(* CODESYS project SeltZVU3.project

Project tree, tasks and I/O mapping:
  Device : Owen SPK1xx, Owen, order no. 023, version 3.5.4.20
    application Application
      libraries: Standard, * (System); CmpSysExec, 1.0.0.2 (Owen); SysTime, * (System); VisuDialogs, * (System); Util, * (System); CAA File, * (CAA Technical Workgroup)
      task MainTask (cyclic, interval t#10ms, priority 1) calls PLC_PRG
      task VISU_TASK (cyclic, interval t#100ms, priority 31) calls VisuElems.Visu_Prg
      task Task_ZAKALKA (cyclic, interval t#10ms, priority 1) calls ZAKALKA
      task READ_WRITE_ZAKALKA_PROG (cyclic, interval t#10ms, priority 1) calls WRITE_PROGRAM_FILE_ON_SD, READ_PROGRAM_FROM_FILE
      task Archivating (cyclic, interval t#10ms, priority 1) calls Archive
      task Task_TransmitingFiles (cyclic, interval t#10ms, priority 1) calls READ_FILE_ON_SD, WRITE_FILE_ON_SD
      task ConnectWithComputer (cyclic, interval t#10ms, priority 1) calls MB_PC
      program PLC_PRG [ST]
      program ClearBuf [ST]
      program DataPrepare [ST]
      program RD_param [ST]
      program READ_PROGRAM_FROM_FILE [ST]: Analyz_str, Find_Symbol
      global variables GVL
      program ZAKALKA [ST]
      program SearchFile [ST]
      text list Modbus_Error_list
      text list Status_v_Rabote
      text list Warning_Text_list
      visualisation Archive_manager
      visualisation Center_indukt
      visualisation KeypadNumpad
      visualisation Modbus_param
      visualisation Regim_choice
      visualisation Zakalka_program
      visualisation Zakalka_work
      program WRITE_PROGRAM_FILE_ON_SD [ST]
      program Archive [ST]: Archivation, make_log_collection, Work_with_Flash
      program WRITE_FILE_ON_SD [ST]
      program READ_FILE_ON_SD [ST]
    SLAVE_COM : Modbus COM, 3S - Smart Software Solutions GmbH, version 3.4.0.0
        settings: DataBits = 8; StopBits = 1; ComPort = 3
      MB_PC : Modbus Serial Device, 3S - Smart Software Solutions GmbH, version 3.5.5.0
          input  Application.buffer_name_file[0] : WORD  // Inputs.Inputs
          input  Application.buffer_name_file[1] : WORD  // Inputs.Inputs
          input  Application.buffer_name_file[2] : WORD  // Inputs.Inputs
          input  Application.buffer_name_file[3] : WORD  // Inputs.Inputs
          input  Application.buffer_name_file[4] : WORD  // Inputs.Inputs
          input  Application.buffer_name_file[5] : WORD  // Inputs.Inputs
          input  Application.buffer_name_file[6] : WORD  // Inputs.Inputs
          input  Application.buffer_name_file[7] : WORD  // Inputs.Inputs
          input  Application.buffer_name_file[8] : WORD  // Inputs.Inputs
          input  Application.buffer_name_file[9] : WORD  // Inputs.Inputs
          input  Application.buffer_name_file[10] : WORD  // Inputs.Inputs
          input  Application.buffer_name_file[11] : WORD  // Inputs.Inputs
          input  Application.buffer_name_file[12] : WORD  // Inputs.Inputs
          input  Application.buffer_name_file[13] : WORD  // Inputs.Inputs
          input  Application.buffer_name_file[14] : WORD  // Inputs.Inputs
          input  Application.buffer_name_file[15] : WORD  // Inputs.Inputs
          input  Application.buffer_name_file[16] : WORD  // Inputs.Inputs
          input  Application.buffer_name_file[17] : WORD  // Inputs.Inputs
          input  Application.buffer_name_file[18] : WORD  // Inputs.Inputs
          input  Application.buffer_name_file[19] : WORD  // Inputs.Inputs
          input  Application.buffer_name_file[20] : WORD  // Inputs.Inputs
          input  Application.buffer_name_file[21] : WORD  // Inputs.Inputs
          input  Application.buffer_name_file[22] : WORD  // Inputs.Inputs
          input  Application.buffer_name_file[23] : WORD  // Inputs.Inputs
          input  Application.buffer_name_file[24] : WORD  // Inputs.Inputs
          input  Application.buffer_wr[0] : WORD  // Inputs.Inputs
          input  Application.buffer_wr[1] : WORD  // Inputs.Inputs
          input  Application.buffer_wr[2] : WORD  // Inputs.Inputs
          input  Application.buffer_wr[3] : WORD  // Inputs.Inputs
          input  Application.buffer_wr[4] : WORD  // Inputs.Inputs
          input  Application.buffer_wr[5] : WORD  // Inputs.Inputs
          input  Application.buffer_wr[6] : WORD  // Inputs.Inputs
          input  Application.buffer_wr[7] : WORD  // Inputs.Inputs
          input  Application.buffer_wr[8] : WORD  // Inputs.Inputs
          input  Application.buffer_wr[9] : WORD  // Inputs.Inputs
          input  Application.buffer_wr[10] : WORD  // Inputs.Inputs
          input  Application.buffer_wr[11] : WORD  // Inputs.Inputs
          input  Application.buffer_wr[12] : WORD  // Inputs.Inputs
          input  Application.buffer_wr[13] : WORD  // Inputs.Inputs
          input  Application.buffer_wr[14] : WORD  // Inputs.Inputs
          input  Application.buffer_wr[15] : WORD  // Inputs.Inputs
          input  Application.buffer_wr[16] : WORD  // Inputs.Inputs
          input  Application.buffer_wr[17] : WORD  // Inputs.Inputs
          input  Application.buffer_wr[18] : WORD  // Inputs.Inputs
          input  Application.buffer_wr[19] : WORD  // Inputs.Inputs
          input  Application.buffer_wr[20] : WORD  // Inputs.Inputs
          input  Application.buffer_wr[21] : WORD  // Inputs.Inputs
          input  Application.buffer_wr[22] : WORD  // Inputs.Inputs
          input  Application.buffer_wr[23] : WORD  // Inputs.Inputs
          input  Application.buffer_wr[24] : WORD  // Inputs.Inputs
          input  Application.buffer_wr[25] : WORD  // Inputs.Inputs
          input  Application.buffer_wr[26] : WORD  // Inputs.Inputs
          input  Application.buffer_wr[27] : WORD  // Inputs.Inputs
          input  Application.buffer_wr[28] : WORD  // Inputs.Inputs
          input  Application.buffer_wr[29] : WORD  // Inputs.Inputs
          input  Application.buffer_wr[30] : WORD  // Inputs.Inputs
          input  Application.buffer_wr[31] : WORD  // Inputs.Inputs
          input  Application.buffer_wr[32] : WORD  // Inputs.Inputs
          input  Application.buffer_wr[33] : WORD  // Inputs.Inputs
          input  Application.buffer_wr[34] : WORD  // Inputs.Inputs
          input  Application.buffer_wr[35] : WORD  // Inputs.Inputs
          input  Application.buffer_wr[36] : WORD  // Inputs.Inputs
          input  Application.buffer_wr[37] : WORD  // Inputs.Inputs
          input  Application.buffer_wr[38] : WORD  // Inputs.Inputs
          input  Application.buffer_wr[39] : WORD  // Inputs.Inputs
          input  Application.buffer_wr[40] : WORD  // Inputs.Inputs
          input  Application.buffer_wr[41] : WORD  // Inputs.Inputs
          input  Application.buffer_wr[42] : WORD  // Inputs.Inputs
          input  Application.buffer_wr[43] : WORD  // Inputs.Inputs
          input  Application.buffer_wr[44] : WORD  // Inputs.Inputs
          input  Application.buffer_wr[45] : WORD  // Inputs.Inputs
          input  Application.buffer_wr[46] : WORD  // Inputs.Inputs
          input  Application.buffer_wr[47] : WORD  // Inputs.Inputs
          input  Application.buffer_wr[48] : WORD  // Inputs.Inputs
          input  Application.buffer_wr[49] : WORD  // Inputs.Inputs
          input  Application.buffer_wr[50] : WORD  // Inputs.Inputs
          input  Application.buffer_wr[51] : WORD  // Inputs.Inputs
          input  Application.buffer_wr[52] : WORD  // Inputs.Inputs
          input  Application.buffer_wr[53] : WORD  // Inputs.Inputs
          input  Application.buffer_wr[54] : WORD  // Inputs.Inputs
          input  Application.buffer_wr[55] : WORD  // Inputs.Inputs
          input  Application.buffer_wr[56] : WORD  // Inputs.Inputs
          input  Application.buffer_wr[57] : WORD  // Inputs.Inputs
          input  Application.buffer_wr[58] : WORD  // Inputs.Inputs
          input  Application.buffer_wr[59] : WORD  // Inputs.Inputs
          input  Application.buffer_wr[60] : WORD  // Inputs.Inputs
          input  Application.buffer_wr[61] : WORD  // Inputs.Inputs
          input  Application.buffer_wr[62] : WORD  // Inputs.Inputs
          input  Application.buffer_wr[63] : WORD  // Inputs.Inputs
          input  Application.buffer_wr[64] : WORD  // Inputs.Inputs
          input  Application.buffer_wr[65] : WORD  // Inputs.Inputs
          input  Application.buffer_wr[66] : WORD  // Inputs.Inputs
          input  Application.buffer_wr[67] : WORD  // Inputs.Inputs
          input  Application.buffer_wr[68] : WORD  // Inputs.Inputs
          input  Application.buffer_wr[69] : WORD  // Inputs.Inputs
          input  Application.buffer_wr[70] : WORD  // Inputs.Inputs
          input  Application.buffer_wr[71] : WORD  // Inputs.Inputs
          input  Application.buffer_wr[72] : WORD  // Inputs.Inputs
          input  Application.buffer_wr[73] : WORD  // Inputs.Inputs
          input  Application.buffer_wr[74] : WORD  // Inputs.Inputs
          input  Application.buffer_wr[75] : WORD  // Inputs.Inputs
          input  Application.buffer_wr[76] : WORD  // Inputs.Inputs
          input  Application.buffer_wr[77] : WORD  // Inputs.Inputs
          input  Application.buffer_wr[78] : WORD  // Inputs.Inputs
          input  Application.buffer_wr[79] : WORD  // Inputs.Inputs
          input  Application.buffer_wr[80] : WORD  // Inputs.Inputs
          input  Application.buffer_wr[81] : WORD  // Inputs.Inputs
          input  Application.buffer_wr[82] : WORD  // Inputs.Inputs
          input  Application.buffer_wr[83] : WORD  // Inputs.Inputs
          input  Application.buffer_wr[84] : WORD  // Inputs.Inputs
          input  Application.buffer_wr[85] : WORD  // Inputs.Inputs
          input  Application.buffer_wr[86] : WORD  // Inputs.Inputs
          input  Application.buffer_wr[87] : WORD  // Inputs.Inputs
          input  Application.buffer_wr[88] : WORD  // Inputs.Inputs
          input  Application.buffer_wr[89] : WORD  // Inputs.Inputs
          input  Application.buffer_wr[90] : WORD  // Inputs.Inputs
          input  Application.buffer_wr[91] : WORD  // Inputs.Inputs
          input  Application.buffer_wr[92] : WORD  // Inputs.Inputs
          input  Application.buffer_wr[93] : WORD  // Inputs.Inputs
          input  Application.buffer_wr[94] : WORD  // Inputs.Inputs
          input  Application.buffer_wr[95] : WORD  // Inputs.Inputs
          input  Application.buffer_wr[96] : WORD  // Inputs.Inputs
          input  Application.buffer_wr[97] : WORD  // Inputs.Inputs
          input  Application.buffer_wr[98] : WORD  // Inputs.Inputs
          input  Application.buffer_wr[99] : WORD  // Inputs.Inputs
          input  Application.buffer_wr[100] : WORD  // Inputs.Inputs
          input  Application.buffer_wr[101] : WORD  // Inputs.Inputs
          input  Application.buffer_wr[102] : WORD  // Inputs.Inputs
          input  Application.buffer_wr[103] : WORD  // Inputs.Inputs
          input  Application.buffer_wr[104] : WORD  // Inputs.Inputs
          input  Application.buffer_wr[105] : WORD  // Inputs.Inputs
          input  Application.buffer_wr[106] : WORD  // Inputs.Inputs
          input  Application.buffer_wr[107] : WORD  // Inputs.Inputs
          input  Application.buffer_wr[108] : WORD  // Inputs.Inputs
          input  Application.buffer_wr[109] : WORD  // Inputs.Inputs
          input  Application.buffer_wr[110] : WORD  // Inputs.Inputs
          input  Application.buffer_wr[111] : WORD  // Inputs.Inputs
          input  Application.buffer_wr[112] : WORD  // Inputs.Inputs
          input  Application.buffer_wr[113] : WORD  // Inputs.Inputs
          input  Application.buffer_wr[114] : WORD  // Inputs.Inputs
          input  Application.buffer_wr[115] : WORD  // Inputs.Inputs
          input  Application.buffer_wr[116] : WORD  // Inputs.Inputs
          input  Application.buffer_wr[117] : WORD  // Inputs.Inputs
          input  Application.buffer_wr[118] : WORD  // Inputs.Inputs
          input  Application.buffer_wr[119] : WORD  // Inputs.Inputs
          input  Application.buffer_wr[120] : WORD  // Inputs.Inputs
          input  Application.WRITE_FILE_ON_SD.size_block : WORD  // Inputs.Inputs
          input  Application.WRITE_FILE_ON_SD.START_STOP_WRITE : WORD  // Inputs.Inputs
          input  Application.READ_FILE_ON_SD.START_STOP_READ : WORD  // Inputs.Inputs
          input  Application.PLC_PRG.SCAN_SD_START_STOP : WORD  // Inputs.Inputs
          input  Application.READ_FILE_ON_SD.RESET_FUNC : WORD  // Inputs.Inputs
          output Application.READ_FILE_ON_SD.SIZE_LR : WORD  // Outputs.Outputs
          output Application.READ_FILE_ON_SD.SIZE_HR : WORD  // Outputs.Outputs
          output Application.buffer[0] : WORD  // Outputs.Outputs
          output Application.buffer[1] : WORD  // Outputs.Outputs
          output Application.buffer[2] : WORD  // Outputs.Outputs
          output Application.buffer[3] : WORD  // Outputs.Outputs
          output Application.buffer[4] : WORD  // Outputs.Outputs
          output Application.buffer[5] : WORD  // Outputs.Outputs
          output Application.buffer[6] : WORD  // Outputs.Outputs
          output Application.buffer[7] : WORD  // Outputs.Outputs
          output Application.buffer[8] : WORD  // Outputs.Outputs
          output Application.buffer[9] : WORD  // Outputs.Outputs
          output Application.buffer[10] : WORD  // Outputs.Outputs
          output Application.buffer[11] : WORD  // Outputs.Outputs
          output Application.buffer[12] : WORD  // Outputs.Outputs
          output Application.buffer[13] : WORD  // Outputs.Outputs
          output Application.buffer[14] : WORD  // Outputs.Outputs
          output Application.buffer[15] : WORD  // Outputs.Outputs
          output Application.buffer[16] : WORD  // Outputs.Outputs
          output Application.buffer[17] : WORD  // Outputs.Outputs
          output Application.buffer[18] : WORD  // Outputs.Outputs
          output Application.buffer[19] : WORD  // Outputs.Outputs
          output Application.buffer[20] : WORD  // Outputs.Outputs
          output Application.buffer[21] : WORD  // Outputs.Outputs
          output Application.buffer[22] : WORD  // Outputs.Outputs
          output Application.buffer[23] : WORD  // Outputs.Outputs
          output Application.buffer[24] : WORD  // Outputs.Outputs
          output Application.buffer[25] : WORD  // Outputs.Outputs
          output Application.buffer[26] : WORD  // Outputs.Outputs
          output Application.buffer[27] : WORD  // Outputs.Outputs
          output Application.buffer[28] : WORD  // Outputs.Outputs
          output Application.buffer[29] : WORD  // Outputs.Outputs
          output Application.buffer[30] : WORD  // Outputs.Outputs
          output Application.buffer[31] : WORD  // Outputs.Outputs
          output Application.buffer[32] : WORD  // Outputs.Outputs
          output Application.buffer[33] : WORD  // Outputs.Outputs
          output Application.buffer[34] : WORD  // Outputs.Outputs
          output Application.buffer[35] : WORD  // Outputs.Outputs
          output Application.buffer[36] : WORD  // Outputs.Outputs
          output Application.buffer[37] : WORD  // Outputs.Outputs
          output Application.buffer[38] : WORD  // Outputs.Outputs
          output Application.buffer[39] : WORD  // Outputs.Outputs
          output Application.buffer[40] : WORD  // Outputs.Outputs
          output Application.buffer[41] : WORD  // Outputs.Outputs
          output Application.buffer[42] : WORD  // Outputs.Outputs
          output Application.buffer[43] : WORD  // Outputs.Outputs
          output Application.buffer[44] : WORD  // Outputs.Outputs
          output Application.buffer[45] : WORD  // Outputs.Outputs
          output Application.buffer[46] : WORD  // Outputs.Outputs
          output Application.buffer[47] : WORD  // Outputs.Outputs
          output Application.buffer[48] : WORD  // Outputs.Outputs
          output Application.buffer[49] : WORD  // Outputs.Outputs
          output Application.buffer[50] : WORD  // Outputs.Outputs
          output Application.buffer[51] : WORD  // Outputs.Outputs
          output Application.buffer[52] : WORD  // Outputs.Outputs
          output Application.buffer[53] : WORD  // Outputs.Outputs
          output Application.buffer[54] : WORD  // Outputs.Outputs
          output Application.buffer[55] : WORD  // Outputs.Outputs
          output Application.buffer[56] : WORD  // Outputs.Outputs
          output Application.buffer[57] : WORD  // Outputs.Outputs
          output Application.buffer[58] : WORD  // Outputs.Outputs
          output Application.buffer[59] : WORD  // Outputs.Outputs
          output Application.buffer[60] : WORD  // Outputs.Outputs
          output Application.buffer[61] : WORD  // Outputs.Outputs
          output Application.buffer[62] : WORD  // Outputs.Outputs
          output Application.buffer[63] : WORD  // Outputs.Outputs
          output Application.buffer[64] : WORD  // Outputs.Outputs
          output Application.buffer[65] : WORD  // Outputs.Outputs
          output Application.buffer[66] : WORD  // Outputs.Outputs
          output Application.buffer[67] : WORD  // Outputs.Outputs
          output Application.buffer[68] : WORD  // Outputs.Outputs
          output Application.buffer[69] : WORD  // Outputs.Outputs
          output Application.buffer[70] : WORD  // Outputs.Outputs
          output Application.buffer[71] : WORD  // Outputs.Outputs
          output Application.buffer[72] : WORD  // Outputs.Outputs
          output Application.buffer[73] : WORD  // Outputs.Outputs
          output Application.buffer[74] : WORD  // Outputs.Outputs
          output Application.buffer[75] : WORD  // Outputs.Outputs
          output Application.buffer[76] : WORD  // Outputs.Outputs
          output Application.buffer[77] : WORD  // Outputs.Outputs
          output Application.buffer[78] : WORD  // Outputs.Outputs
          output Application.buffer[79] : WORD  // Outputs.Outputs
          output Application.buffer[80] : WORD  // Outputs.Outputs
          output Application.buffer[81] : WORD  // Outputs.Outputs
          output Application.buffer[82] : WORD  // Outputs.Outputs
          output Application.buffer[83] : WORD  // Outputs.Outputs
          output Application.buffer[84] : WORD  // Outputs.Outputs
          output Application.buffer[85] : WORD  // Outputs.Outputs
          output Application.buffer[86] : WORD  // Outputs.Outputs
          output Application.buffer[87] : WORD  // Outputs.Outputs
          output Application.buffer[88] : WORD  // Outputs.Outputs
          output Application.buffer[89] : WORD  // Outputs.Outputs
          output Application.buffer[90] : WORD  // Outputs.Outputs
          output Application.buffer[91] : WORD  // Outputs.Outputs
          output Application.buffer[92] : WORD  // Outputs.Outputs
          output Application.buffer[93] : WORD  // Outputs.Outputs
          output Application.buffer[94] : WORD  // Outputs.Outputs
          output Application.buffer[95] : WORD  // Outputs.Outputs
          output Application.buffer[96] : WORD  // Outputs.Outputs
          output Application.buffer[97] : WORD  // Outputs.Outputs
          output Application.buffer[98] : WORD  // Outputs.Outputs
          output Application.buffer[99] : WORD  // Outputs.Outputs
          output Application.buffer[100] : WORD  // Outputs.Outputs
          output Application.buffer[101] : WORD  // Outputs.Outputs
          output Application.buffer[102] : WORD  // Outputs.Outputs
          output Application.buffer[103] : WORD  // Outputs.Outputs
          output Application.buffer[104] : WORD  // Outputs.Outputs
          output Application.buffer[105] : WORD  // Outputs.Outputs
          output Application.buffer[106] : WORD  // Outputs.Outputs
          output Application.buffer[107] : WORD  // Outputs.Outputs
          output Application.buffer[108] : WORD  // Outputs.Outputs
          output Application.buffer[109] : WORD  // Outputs.Outputs
          output Application.buffer[110] : WORD  // Outputs.Outputs
          output Application.buffer[111] : WORD  // Outputs.Outputs
          output Application.buffer[112] : WORD  // Outputs.Outputs
          output Application.buffer[113] : WORD  // Outputs.Outputs
          output Application.buffer[114] : WORD  // Outputs.Outputs
          output Application.buffer[115] : WORD  // Outputs.Outputs
          output Application.buffer[116] : WORD  // Outputs.Outputs
          output Application.buffer[117] : WORD  // Outputs.Outputs
          output Application.buffer[118] : WORD  // Outputs.Outputs
          output Application.buffer[119] : WORD  // Outputs.Outputs
          output Application.buffer[120] : WORD  // Outputs.Outputs
          output Application.buffer[121] : WORD  // Outputs.Outputs
          output Application.buffer[122] : WORD  // Outputs.Outputs
          output Application.buffer[123] : WORD  // Outputs.Outputs
          output Application.buffer[124] : WORD  // Outputs.Outputs
          output Application.WRITE_FILE_ON_SD.CycleWriteDone : WORD  // Outputs.Outputs
          output Application.FileError : WORD  // Outputs.Outputs
          output Application.READ_FILE_ON_SD.RESET_SUC : BOOL  // Outputs.Outputs.Bit0
          output Application.READ_FILE_ON_SD.cnt_cycle : WORD  // Outputs.Outputs
          unmapped channels: Inputs, Outputs
    Modbus_COM : Modbus COM, 3S - Smart Software Solutions GmbH, version 3.4.0.0
        settings: DataBits = 8; StopBits = 1; ComPort = 2
      Modbus_Master_COM_Port : Modbus Master, COM Port, 3S - Smart Software Solutions GmbH, version 3.5.5.0
          settings: Transmission = 'RTU'; ResponseTimeout = 500; TimeBetweenFrames = 50; Auto-restart communication = TRUE
        Modbus_Slave_Atxmega128 : Modbus Slave, COM Port, 3S - Smart Software Solutions GmbH, version 3.5.4.0
            settings: SlaveAddress = 9; ResponseTimeout = 500; UseExtendedFunctionCodes = TRUE; Channel7.Function Code = 3; Channel7.Read Offset = 16#0000; Channel7.Read Length = 51; Channel7.Write Offset = 0; Channel7.Write Length = 0; Channel7.Cycle Time = 500; To_Atxmega_KN_NACHALO.Function Code = 16; To_Atxmega_KN_NACHALO.Read Offset = 0; To_Atxmega_KN_NACHALO.Read Length = 0; To_Atxmega_KN_NACHALO.Write Offset = 16#0032; To_Atxmega_KN_NACHALO.Write Length = 1; To_Atxmega_KN_NACHALO.Cycle Time = 500; Channel 2.Function Code = 4; Channel 2.Read Offset = 16#0000; Channel 2.Read Length = 23; Channel 2.Write Offset = 0; Channel 2.Write Length = 0; Channel 2.Cycle Time = 500; Channel 3.Function Code = 16; Channel 3.Read Offset = 0; Channel 3.Read Length = 0; Channel 3.Write Offset = 16#0001; Channel 3.Write Length = 12; Channel 3.Cycle Time = 100; Channel 6.Function Code = 6; Channel 6.Read Offset = 0; Channel 6.Read Length = 0; Channel 6.Write Offset = 16#0000; Channel 6.Write Length = 1; Channel 6.Cycle Time = 100; Channel 5.Function Code = 16; Channel 5.Read Offset = 0; Channel 5.Read Length = 0; Channel 5.Write Offset = 16#0033; Channel 5.Write Length = 123; Channel 5.Cycle Time = 100
            input  Application.PLC_PRG.DY_start : WORD  // Channel7.Channel7
            input  Application.ZAKALKA.opros_DY_kn_nachalo : BOOL  // Channel7.Channel7.Bit0
            output Application.PLC_PRG.DY_kn_nachalo : BOOL  // To_Atxmega_KN_NACHALO.To_Atxmega_KN_NACHALO.Bit0
            input  Application.PLC_PRG.PORTKH : WORD  // Channel 2.Channel 2
            input  Application.PLC_PRG.PORTCF : WORD  // Channel 2.Channel 2
            input  Application.PLC_PRG.WarningText_mod : WORD  // Channel 2.Channel 2
            input  Application.t_prog_LCD : WORD  // Channel 2.Channel 2
            input  Application.W_schet_vat : WORD  // Channel 2.Channel 2
            input  Application.zona : WORD  // Channel 2.Channel 2
            input  Application.P_ind : WORD  // Channel 2.Channel 2
            input  Application.T_rad_max : WORD  // Channel 2.Channel 2
            input  Application.zona_reg : WORD  // Channel 2.Channel 2
            input  Application.n_nagrev : WORD  // Channel 2.Channel 2
            input  Application.i_t_regim : WORD  // Channel 2.Channel 2
            input  Application.Frec_LCD_point : WORD  // Channel 2.Channel 2
            input  Application.U_pit_max : WORD  // Channel 2.Channel 2
            input  Application.tekyheePosition_lcd : WORD  // Channel 2.Channel 2
            input  Application.I_lcd : WORD  // Channel 2.Channel 2
            input  Application.zadachaPosition_lcd : WORD  // Channel 2.Channel 2
            output Application.PLC_PRG.UP_DOWN : WORD  // Channel 3.Channel 3
            output Application.DistRegim : WORD  // Channel 3.Channel 3
            output Application.PLC_PRG.MB_4_20_kanal_1 : WORD  // Channel 3.Channel 3
            output Application.PLC_PRG.MB_4_20_kanal_2 : WORD  // Channel 3.Channel 3
            output Application.ZAKALKA.zakalka_nachalo : WORD  // Channel 3.Channel 3
            output Application.ZAKALKA.rotation_on : BOOL  // Channel 3.Channel 3.Bit0
            output Application.ZAKALKA.spreer_prednagrev : BOOL  // Channel 3.Channel 3.Bit0
            output Application.ZAKALKA.diagnostik : BOOL  // Channel 3.Channel 3.Bit0
            output Application.ZAKALKA.OTPUSK : BOOL  // Channel 3.Channel 3.Bit0
            output Application.L_peremesh_ohl : WORD  // Channel 3.Channel 3
            output Application.PLC_PRG.b_req_start_stop : BIT  // Channel 6
            output Application.PLC_PRG.CMD_start : ARRAY[0..0] OF WORD  // Channel 6
            output Application.PLC_PRG.Req_WR_Params : BIT  // Channel 5
            output Application.PLC_PRG.Buffer : ARRAY[0..122] OF WORD  // Channel 5
            unmapped channels: Channel7, To_Atxmega_KN_NACHALO, Channel 2, Channel 3
        Modbus_Slave_MY110 : Modbus Slave, COM Port, 3S - Smart Software Solutions GmbH, version 3.5.4.0
            settings: SlaveAddress = 16; ResponseTimeout = 500; UseExtendedFunctionCodes = TRUE; Channel 0.Function Code = 15; Channel 0.Read Offset = 0; Channel 0.Read Length = 0; Channel 0.Write Offset = 16#0000; Channel 0.Write Length = 8; Channel 0.Cycle Time = 250
            output Application.PLC_PRG.ZAGIM_UP : BOOL  // Channel 0.Channel 0.Bit0
            output Application.PLC_PRG.ZAGIM_DOWN : BOOL  // Channel 0.Channel 0.Bit1
            output Application.PLC_PRG.CENTER_DOWN : BOOL  // Channel 0.Channel 0.Bit2
            output Application.PLC_PRG.CENTER_UP : BOOL  // Channel 0.Channel 0.Bit3
            output Application.PLC_PRG.DET_CIRCLE_ON : BOOL  // Channel 0.Channel 0.Bit4
            output Application.PLC_PRG.SPREER_ON : BOOL  // Channel 0.Channel 0.Bit5
            output Application.PLC_PRG.CENTER_LEFT : BOOL  // Channel 0.Channel 0.Bit6
            output Application.PLC_PRG.CENTER_RIGHT : BOOL  // Channel 0.Channel 0.Bit7
            unmapped channels: Channel 0
  text list GlobalTextList
  text list NachaloVerhNiz
*)

// Device/Application/GVL
VAR_GLOBAL
	ProgramFiles:STRING(255):='/mnt/ufs/media/mmcblk0p1/ProgramFiles/';
	ArchiveFiles:STRING(255):='/mnt/ufs/media/mmcblk0p1/Archive/';		
	nomer_zoni: ARRAY [1..20] OF INT;
	zona_rabochaya: USINT := 1;	
	
	(*Датчики*)
	PORTK: BYTE;
	PORTH: BYTE;
	PORTC: BYTE;
	PORTF: BYTE;
	
	WarningText: WORD := 1;
	t_prog_LCD: WORD;
	W_schet_vat: WORD;
	zona : WORD;
	P_ind: WORD;
	T_rad_max: WORD;
	zona_reg: WORD;
	n_nagrev: WORD;
	R_ind_lcd: WORD; 
	i_t_regim: WORD := 3;
	DistRegim: WORD;
	DY_gotovn : BOOL;
	Frec_LCD: WORD;
	U_pit_max: WORD;
	U_pit_min: WORD;
 	tekyheePosition_lcd: WORD;
	Frec_LCD_point:WORD;
	h_faza:WORD;
	I_lcd:WORD;
	zadachaPosition_lcd: WORD;
	
	rotation_on: BOOL; 
	
	buffer: ARRAY[0..125] OF WORD;
	buffer_name_file: ARRAY [0..24] OF WORD;
	buffer_wr: ARRAY[0..120] OF WORD;
	
	FileError: INT;//Ошибка при записи файла по модбасу
	ExError	: BOOL;
	StrError : STRING(255);
	READING: BOOL;
	WRITING: BOOL;
	RESET_ERROR:BOOL;
	
(*	OTPUSK_P_nachaln_nagrev: ARRAY [1..10] OF INT;
	OTPUSK_t_nachaln_nagrev: ARRAY [1..10] OF INT;
	OTPUSK_P_nagrev: ARRAY [1..10] OF INT;
	OTPUSK_V_peremeshenia: ARRAY [1..10] OF BYTE;
	OTPUSK_t_freeze: ARRAY [1..10] OF INT;*)
	
END_VAR

VAR_GLOBAL PERSISTENT RETAIN
	chislo_zon: WORD := 1;
//	Nachalo: INT;//Зачем убрал из параметров для хранения в ПЗУ ?	
	P_nachaln_nagrev: ARRAY [1..20] OF INT;//Мощность на преднагрев
	t_nachaln_nagrev: ARRAY [1..20] OF INT;//Время а преднагрев
	P_nagrev: ARRAY [1..20] OF INT;//Мощность в движени
	L_peremeshenia: ARRAY [1..20] OF INT;//Длиназоны
	V_peremeshenia: ARRAY [1..20] OF INT;//Сорость пермщеия
	t_freeze: ARRAY [1..20] OF INT;//Вемя охлаждения
	L_to_next_zone: ARRAY [1..20] OF INT;//Растояние до слдующейзоны
	L_peremesh_ohl: WORD;
END_VAR

// Device/Application/PLC_PRG
PROGRAM PLC_PRG

VAR_INPUT
	ReqStart : BOOL := FALSE; //Запрос на старт при нажатие кнопок старт = 1 после отправки запроса = 0
	Req_WR_Params : BOOL := FALSE; //запрос на передачу параметров в МК
	Req_OverWriting_param : BOOL := FALSE;
	DY_start: WORD;//отображает состояние кнопок старт/стоп и состояние МК
	CMD_start: WORD;//1-Старт 0-Стоп
	Req_START_STOP: BOOL;//Запрос на передачу команды старт/стоп
	DY_kn_nachalo: BOOL := FALSE; //кнопка начало 0-неактивна 1-актив
END_VAR

VAR
	Timer_Req_WR_params:TON;
	Timer_Inc_Speed:TON;
	TMR_START:TON;
	b_req_start_stop:BOOL;//Тригер для передачи команды старт стоп
	MB_4_20_kanal_2 : INT:=7000;//Скорость вращения нижнего центра
	MB_4_20_kanal_1 : INT:=7000;//Скорость перемещения индуктора/детали	
	
	PORTKH: WORD;
	PORTCF: WORD;
	ReqStop : BOOL := FALSE; //Запрос на стоп при нажатие кнопок стоп = 1 после отправки запроса = 0
	
	UP_DOWN : WORD := 0; // верх вниз 0-стоп 1-в верх 2-в низ
	
 
	START: BOOL := FALSE; //старт установки
	STOP: BOOL := TRUE; //стоп установки
	
	CENTER_UP: BOOL;
	CENTER_DOWN: BOOL;
	CENTER_LEFT: BOOL;
	CENTER_RIGHT: BOOL;
	ZAGIM_UP: BOOL;
	ZAGIM_DOWN: BOOL;
	DET_CIRCLE_ON: BOOL;	//вкл вращение
	DET_CIRCLE_SPIN: BOOL; //вкл регулирование скорости
	DET_CIRCLE_SPEED: WORD; //скорость вращения детали
	SPREER_ON: BOOL;
	
	Buffer : ARRAY[0..122] OF WORD;
	cmpl: BOOL;
	err: INT;
	TimeOut : TIME:=T#300MS;
	DataSize : WORD;
	Connect : BOOL :=FALSE;
	master : BYTE := 3;
	CNT_REG : BYTE;
	
	(*Входные параметры*)
	in1: BOOL;
	in2: BOOL; 
	in3: BOOL;//Датчик низа
	in4: BOOL;
	in5: BOOL;
	in6: BOOL;//Датчик верха
	in7: BOOL;
	in8: BOOL;
	in9: BOOL;
	in10: BOOL;//Кнопка начало
	in11: BOOL;
	
	TEMP  : WORD;  
	(*конец входные параметры*)
	
	Button: WORD;
	ButAddr: WORD;
	
	WarningText_mod: WORD;
	Butt_UP: BOOL;
	Butt_DOWN: BOOL;
	
	//Время
	result_time: UDINT;
	time_dword: DWORD;
	time_of_st: DATE_AND_TIME;
	
	Symbols: ARRAY[0..4] OF BYTE;
	stroka:STRING;
	p_str:POINTER TO BYTE;
	i:BYTE;
	
	(*Работа с файловой системой*)
	SCAN_SD_START_STOP:WORD;
	ErrorModbus_Atxmega: IoDrvModbus.MB_ErrorCodes;
	ErrorModbus_MY110: INT;
END_VAR

PORTK := WORD_TO_BYTE(SHR(PORTKH,8));
PORTH := WORD_TO_BYTE(PORTKH);
PORTC := WORD_TO_BYTE(SHR(PORTCF,8));
PORTF := WORD_TO_BYTE(PORTCF);
in1 := NOT(GVL.PORTK.4);
in2 := GVL.PORTK.5;
in3 := GVL.PORTK.6;
in4 := GVL.PORTK.7;
in5 := GVL.PORTH.3;
in6 := GVL.PORTH.2;
in7 := GVL.PORTC.2;
in8 := GVL.PORTC.3;
in9 := GVL.PORTC.4;
in10:= GVL.PORTC.5;
in11:= GVL.PORTF.6;

IF CMD_start=DY_start=1 THEN
	Req_START_STOP:=FALSE;
END_IF

TMR_START(IN:=Req_START_STOP,PT:=T#50MS);
IF TMR_START.Q THEN
	TMR_START(IN:=FALSE);
	b_req_start_stop:=NOT(b_req_start_stop);
END_IF

Timer_Req_WR_params(IN:=DY_kn_nachalo OR Req_OverWriting_param, PT:=T#200MS , Q=> , ET=> );
IF Timer_Req_WR_params.Q THEN //(DY_kn_nachalo OR Req_OverWriting_param) AND (cnt_timer>30)THEN
	DataPrepare(chislo_zon:=GVL.chislo_zon,P_nachaln_nagrev:=GVL.P_nachaln_nagrev,t_nachaln_nagrev:=GVL.t_nachaln_nagrev,P_nagrev:=GVL.P_nagrev,V_peremeshenia:=GVL.V_peremeshenia,L_peremeshenia:=GVL.L_peremeshenia,L_to_next_zone:=GVL.L_to_next_zone,t_freeze:=GVL.t_freeze, Buffer=>Buffer);
	Timer_Req_WR_params(IN:=FALSE);
//	DY_kn_nachalo:=FALSE;
	Req_OverWriting_param:=FALSE;
	Req_WR_Params:=TRUE;
END_IF

Timer_Inc_Speed(IN:=((UP_DOWN=2) OR (UP_DOWN=1)), PT:=T#100MS , Q=> , ET=> );
IF Timer_Inc_Speed.Q THEN //(DY_kn_nachalo OR Req_OverWriting_param) AND (cnt_timer>30)THEN
	Timer_Inc_Speed(IN:=FALSE);
	IF MB_4_20_kanal_1  + 100 >= 20000 THEN
		MB_4_20_kanal_1:=20000;	
	ELSE
		MB_4_20_kanal_1:=MB_4_20_kanal_1+100;	
	END_IF
END_IF

IF UP_DOWN=0 THEN
	MB_4_20_kanal_1:=7000;
END_IF

IF dy_start = 1 THEN
	VisuElems.CurrentVisu:='Zakalka_work';
END_IF

IF (dy_start = 0) AND (VisuElems.CurrentVisu = 'Zakalka_work') THEN
	VisuElems.CurrentVisu := 'Zakalka_program';
END_IF

time_dword:=SysTimeRtcGet(pResult:=result_time );
time_of_st:=DWORD_TO_DT(time_dword);

ErrorModbus_Atxmega := Modbus_Slave_Atxmega128.byModbusError;
ErrorModbus_MY110 := Modbus_Slave_MY110.byModbusError;

END_PROGRAM

// Device/Application/DataPrepare
PROGRAM DataPrepare
VAR_INPUT
	chislo_zon: WORD;
	P_nachaln_nagrev: ARRAY [1..20] OF INT;
	t_nachaln_nagrev: ARRAY [1..20] OF INT;
	P_nagrev: ARRAY [1..20] OF INT;
	V_peremeshenia: ARRAY [1..20] OF INT;
	L_peremeshenia: ARRAY [1..20] OF INT;
	L_to_next_zone: ARRAY [1..20] OF INT;
	t_freeze: ARRAY [1..20] OF INT;
END_VAR

VAR_OUTPUT
	Buffer: ARRAY[0..122] OF WORD;
END_VAR

VAR
	TEMP: INT;
	Counter: INT;
	index: INT;
	knopka_nachalo: BYTE :=1;
END_VAR

index:=0;
Buffer[index]:= chislo_zon;
index:=index+1;
	
FOR Counter:=(1+ZAKALKA.shift_otpusk) TO (chislo_zon+ZAKALKA.shift_otpusk) BY 1 DO
	Buffer[index]:= t_nachaln_nagrev[Counter];
	index:=index+1;
	
	Buffer[index]:= p_nachaln_nagrev[Counter];
	index:=index+1;
	
	Buffer[index]:= V_peremeshenia[Counter];
	index:=index+1;
	

	Buffer[index]:= L_peremeshenia[Counter-ZAKALKA.shift_otpusk];
	index:=index+1;


	Buffer[index]:= P_nagrev[Counter];
	index:=index+1;
	
	
	Buffer[index]:= t_freeze[Counter];
	index:=index+1;
	
	Buffer[index]:= L_to_next_zone[Counter-ZAKALKA.shift_otpusk];
	index:=index+1;
END_FOR

END_PROGRAM

// Device/Application/ZAKALKA
PROGRAM ZAKALKA
VAR
Zakalochniy_cikl: INT;
stage: INT := 1;	
AutoCicleFinish:WORD;

Zakalka_otpusk_active: BOOL := TRUE; //выбран ярлык редактирования отпуска
L_between_stels: BOOL := TRUE;
i_zona: USINT := 1; //заполнитель кнопки зона
OTPUSK: BOOL;//Запуск отпуска


shift_otpusk: INT;
Zakalka_last_zona: BOOL;
color_indukt: DWORD;

pressed_find_prog:BOOL;//true когда нажата кнопка найти программу
pressed_create_new_prog:BOOL;
enter_value:BOOL;//true - при закрытии клавы по кнопке OK
SearchThroughArray: STRING;//Имя файла для поиска существующей программы закалки
new_prog: STRING;//Имя файла для новой программы 
result_prog: ARRAY [1..10] OF STRING(255);//Результаты поиска
	i_result_prog: INT :=1;//Активный размер масива result_prog
enter_prog: INT:=1;//Индекс выбранной программы в массиве result_prog
buf_enter_prog : INT:=1;//Предыдущее значение enter_prog
test_ok: BOOL :=FALSE;
	opros_DY_kn_nachalo: BOOL;
update_drop_list:BOOL;
	buf_size_list:INT;//предыдущая длина списка найденных файлов
END_VAR

VAR_INPUT
	Otpusk_on: BOOL;//отпуск включен
	Zakalka_on: BOOL:=TRUE;
 	spreer_prednagrev: BOOL;
	diagnostik: BOOL:=TRUE;
	rotation_on: BOOL:=TRUE; 
	
	zakalka_nachalo: INT;
END_VAR
VAR_OUTPUT

END_VAR

IF PLC_PRG.DY_start=1 THEN
	Archive.arch_en:=TRUE;
ELSE	
	Archive.arch_en:=FALSE;
END_IF

IF (PLC_PRG.DY_kn_nachalo) AND (opros_DY_kn_nachalo = TRUE) THEN
	PLC_PRG.DY_kn_nachalo := FALSE;
END_IF

IF (Otpusk_on <> TRUE) THEN
	Zakalka_otpusk_active := TRUE;
ELSE
	IF (ZAKALKA.Zakalka_on <> TRUE) THEN
	Zakalka_otpusk_active := FALSE;
	END_IF
END_IF

IF (zona_rabochaya = chislo_zon) THEN
	Zakalka_last_zona := TRUE;
ELSE
	Zakalka_last_zona := FALSE;
END_IF


IF PLC_PRG.DY_start = 0  AND ((ZAKALKA.stage <> 3 AND ZAKALKA.stage <> 2) OR (PLC_PRG.WarningText_mod = 53)) THEN
	ZAKALKA.stage := 0;
	
	IF (ZAKALKA.Zakalka_on) AND (ZAKALKA.Otpusk_on = FALSE) THEN //цикл закалка без отпуска
		ZAKALKA.Zakalochniy_cikl := 1;
		shift_otpusk := 0;
		OTPUSK := FALSE;
	END_IF
	
	IF (ZAKALKA.Zakalka_on = FALSE) AND (ZAKALKA.Otpusk_on) THEN //цикл отпуск без закалки
		ZAKALKA.Zakalochniy_cikl := 2;
		shift_otpusk := 10;
		OTPUSK := TRUE;
	END_IF
	
	IF (ZAKALKA.Zakalka_on) AND (ZAKALKA.Otpusk_on) THEN		//цикл закалка с отпуском
		ZAKALKA.Zakalochniy_cikl := 3;
		shift_otpusk := 0;
		OTPUSK := FALSE;
	END_IF
		PLC_PRG.Req_WR_Params := FALSE;
		PLC_PRG.Req_OverWriting_param := TRUE;
END_IF

IF PLC_PRG.DY_start = 1  AND ZAKALKA.stage = 0 THEN
	ZAKALKA.stage := 1;
END_IF

//включения отпуска в момент основного нагрева
IF (PLC_PRG.DY_start = 1) AND (ZAKALKA.Zakalochniy_cikl = 3) AND (zona = chislo_zon) THEN
	IF (ZAKALKA.stage = 3) THEN
//			 OTPUSK := TRUE;
			 Zakalka.stage := 4;
	END_IF
	IF (ZAKALKA.stage = 1) THEN

			 Zakalka.stage := 2;
	END_IF

//ELSE 
//	shift_otpusk := 0;
END_IF



//запуск отпуска после отработки основного цикла
IF PLC_PRG.DY_start = 0 THEN//закончен автоцикл закалки
	IF ZAKALKA.stage = 2 THEN 
		shift_otpusk := 10;
		OTPUSK := TRUE;
		PLC_PRG.Req_WR_Params := FALSE;
		PLC_PRG.Req_OverWriting_param := TRUE;
		IF ((PLC_PRG.in6 = 0) OR (PLC_PRG.in3 = 0)) THEN
			PLC_PRG.Req_START_STOP:=TRUE;//Автоматический запуск отпуска
			PLC_PRG.CMD_start:=1;
			ZAKALKA.stage := 3;
//			shift_otpusk := 0;
			//OTPUSK := FALSE;
		END_IF
	END_IF
ELSE 
//	OTPUSK := FALSE;
END_IF





IF (chislo_zon > 1) AND (zona < chislo_zon) THEN
	ZAKALKA.L_between_stels := FALSE;
ELSE
	ZAKALKA.L_between_stels := TRUE;	
END_IF

IF zona_rabochaya > chislo_zon THEN
	zona_rabochaya := 1;
END_IF

WHILE (ZAKALKA.i_zona <> 11) DO
	nomer_zoni[ZAKALKA.i_zona] := ZAKALKA.i_zona;
	ZAKALKA.i_zona := ZAKALKA.i_zona + 1; 	
END_WHILE


IF pressed_find_prog THEN//Click на найти программу
	IF enter_value THEN//ввод через клавиаутуру закончен
	pressed_find_prog:=FALSE;
	enter_value:=FALSE;
//	i_result_prog := 1;

	SearchFile(temple_name:=SearchThroughArray, dir:=ProgramFiles, get_list:=FALSE, file_list:='list.txt', list=>result_prog, size_list=>i_result_prog);
	IF i_result_prog=0 THEN
		result_prog[1]:='Not Found';
		i_result_prog:=1;
	END_IF
	READ_PROGRAM_FROM_FILE(name_file_prog:=result_prog[enter_prog], begin:=TRUE);
	enter_prog := 1;	
	END_IF
END_IF

IF pressed_create_new_prog THEN
	IF enter_value THEN//ввод через клавиаутуру закончен
		pressed_create_new_prog:=FALSE;
		enter_value:=FALSE;
		WRITE_PROGRAM_FILE_ON_SD(name_file:=new_prog, wr:=TRUE);
	END_IF
END_IF

IF enter_prog<>buf_enter_prog THEN
	READ_PROGRAM_FROM_FILE(name_file_prog:=result_prog[enter_prog], begin:=true);
	buf_enter_prog:=enter_prog;
END_IF

CASE i_t_regim OF
	0: color_indukt := 16#D77D31;
	1: color_indukt := 16#FF0000;
	2: color_indukt := 16#6600FF;
	4: color_indukt := 16#999999;
END_CASE

END_PROGRAM

// Device/Application/Archive
PROGRAM Archive
VAR_INPUT
	arch_en				: BOOL;
END_VAR
VAR
	(*Архив*)
	log_message			: STRING(255);
	check_mount			: BOOL;
	log_write_done		: BOOL:=TRUE;
	unmount				: BOOL;
	memory_all 			: STRING ;
	memory_used 		: WSTRING ;
	memory_percent 		: REAL;
	
	my_mes				: STRING(255);
	old_mounth			: UINT;
	mounth_changed		: BOOL;
	tr_Mounth			: R_trig;
	arch_case			: INT := 100;
	arc_case			: INT;
	arc_err				: BOOL;
	log_state			: INT;
	log_open			: FILE.Open;
	log_write			: file.write;
	get_log_pos			: FILE.GetPos;
	get_log_size		: FILE.GetSize;
	set_log_pos			: FILE.SetPos;
	log_size			: UDINT;
	Log_write_wait		: TON;
	Log_file_close		: FILE.Close;
	mounted				: BOOL;
	w					: STRING;
	sys3				: sysExecute2;
	time_of_st			: DATE_AND_TIME;
	linear				: LIN_TRAFO;
	i					: BYTE;
	memory_trafo		: LIN_TRAFO;
	memory_free_rotate	: REAL;
	scan_flash			: BOOL;
	in_system			: BOOL;
	reset_in_sys		: R_TRIG;
	trig_to_find_info	: R_TRIG;
	take_info			: BOOL;
	flash_info			: ARRAY [0..5] OF STRING [25];
	anti_empty			: STRING;

	rescan_timer		: TON;
	info_trig			: F_TRIG;
	arch_timer			: TON;
	transmit_en         : BOOL;
	
	Arch_timout			: DWORD:=1;
	scan_timer			: INT;
	scan_timout			: TIME;
	can_arch			: BOOL;
	
	en_arch_P		: BOOL;
	en_arch_I		: BOOL;
	en_arch_Z		: BOOL;
	en_arch_H		: BOOL;
	
	point_byte: POINTER TO ARRAY [0..255] OF BYTE;
	j: INT;
	
	
	
	buffer: ARRAY [0..1000] OF BYTE;
	buffer_1: ARRAY [0..1000] OF BYTE;
	
	size_str:INT;
	k: INT;
	mylen: INT;
	arc_name_need: BOOL;
	unmount_F_trig: F_TRIG;
	
	may_in_sys: BOOL;
	um_ton: Ton;
	iterator: UDINT;
	
	memory_all_word: dWORD;
END_VAR

Work_with_Flash();

ACTION Archivation:
// /mnt/ufs/media/mmcblk0p1/ SD
// /mnt/ufs/media/sda1/ FLASH

IF NOT log_write_done AND CAN_ARCH THEN

	CASE log_state OF
		0:
		FOR j:=0 TO k DO 
			buffer[j]:=buffer_1[j];
			IF buffer[j] = 35 THEN
				buffer[j]:=0;
			END_IF
			BUFFER_1[j]:=0;
		END_FOR
		k:=0;		
		
		get_log_size(
			xExecute:= TRUE, 
			xDone=> , 
			xBusy=> , 
			xError=> , 
			sFileName:=concat(ArchiveFiles,concat('log','.csv')) , 
			eError=> , 
			szSize=>log_size );
			
			IF get_log_size.xDone OR get_log_size.eError=file.ERROR.NOT_EXIST THEN
				get_log_size(xExecute:= FALSE);
				log_state:=1;
			END_IF

		1:		
		log_open(
		xExecute:=TRUE , 
		xDone=> , 
		xBusy=> , 
		xError=> , 

		sFileName:=concat(ArchiveFiles,concat('log','.csv')), 
		eFileMode:=SEL(log_size<>0,file.MODE.MWRITE,file.MODE.MAPPD) , 
		xExclusive:=, 
		eError=> , 
		hFile=> );
		
		IF log_open.xDone AND NOT log_open.xError THEN
			log_state:=2;
		END_IF
		
		2:
		set_log_pos(
			xExecute:=TRUE , 
			xDone=> , 
			xBusy=> , 
			xError=> , 
			hFile:=log_open.hFile , 
			udiPos:=log_size , 
			eError=> );
		
		IF set_log_pos.xDone THEN
			log_state:=3;
			IF log_size =0 THEN
				log_message:= 'Дата;Время,сек;Мощность,кВт;Ток,А;Зона;Частота,кГц;Температура,°C$N';
				mylen:=len(log_message);
				arc_name_need:=TRUE;//надо заархивировать имя
			END_IF
		END_IF
			
		3:	
		log_write(
			xExecute:=TRUE , 
			xAbort:= , 
			udiTimeOut:=100000 , 
			xDone=> , 
			xBusy=> , 
			xError=> , 
			xAborted=> , 
			hFile:=log_open.hFile , 
			pBuffer:=SEL(arc_name_need,ADR(BUFFER),ADR(log_message)) ,
			szSize:= SEL(arc_name_need,size_str,mylen), 
			eError=> );
			
		//Log_write_wait(IN:=TRUE , PT:=T#10S , Q=> , ET=> );
		IF log_write.xDone (*AND Log_write_wait.Q*) THEN
			IF NOT log_write.xError THEN
				IF NOT arc_name_need THEN
			
					Log_write_wait(in:=FALSE);
					set_log_pos(xExecute:=FALSE);
					log_write(xExecute:=FALSE);
					log_message:='';
					log_state:=4;
					FOR j:=0 TO 990 DO
						BUFFER[j]:=0;
					END_FOR
					//k:=0;
				ELSE
					log_write(xExecute:=FALSE);
					arc_name_need:=false;
				END_IF
				iterator:=iterator+log_write.szSize;
				size_str:=0;
			END_IF
			
		END_IF
		
		4:
		Log_file_close(
			xExecute:=TRUE , 
			xDone=> , 
			xBusy=> , 
			xError=> , 
			hFile:=log_open.hFile , 
			eError=> );
		
	IF Log_file_close.xDone THEN
		log_open(xexecute:=FALSE);
		Log_file_close(xexecute:=FALSE);
		log_state:=5;
	END_IF
		
		
		5:
		sysExecute(sys_command:='sync');
		
		IF iterator>1024*1024 THEN
			sysExecute(sys_command:='echo 3 > /proc/sys/vm/drop_caches');(*сброс кэша для освобождения оперативки*)
			iterator:=0;
		END_IF
		
		log_write_done:=TRUE;
		log_state:=0;
		
		
	END_CASE

END_IF
END_ACTION

ACTION make_log_collection:
(*cбор данных к архивации*)
IF arch_timer.Q THEN
	// тут вставить данные на архивацию.
	log_message:=concat(mid(DT_TO_STRING(plc_prg.time_of_st),len(DT_TO_STRING(plc_prg.time_of_st))-2,3),';'); //Дата 2015-10-12 20:41:59
	log_message:=concat(log_message, concat(WORD_TO_STRING(GVL.t_prog_LCD),';'));//Время работы установки t_prog_LCD
	log_message:=concat(log_message, concat(WORD_TO_STRING(GVL.P_ind),';'));//Выдаваемая мощность
	log_message:=concat(log_message, concat(WORD_TO_STRING(GVL.I_lcd),';'));//Ток индуктора
	log_message:=concat(log_message, concat(concat(WORD_TO_STRING(GVL.zona_reg),concat(',',mid(WORD_TO_STRING(GVL.h_faza),1,1))),';'));//Зона регулирования
	log_message:=concat(log_message, concat(REAL_TO_STRING(GVL.Frec_LCD_point/10.0),';'));//Частота
	log_message:=concat(log_message, concat(REAL_TO_STRING(GVL.T_rad_max),';'));//Температура
	log_message:=concat(log_message, '$N');//Перевод на следующую строку
			
	point_byte:=ADR(log_message);
	FOR J:=0 TO len(log_message) DO
		buffer_1[k] := point_byte^[J];
		//point_byte:=point_byte+1;
		size_str:=size_str+1;
		k:=k+1;
		IF k>=990 THEN
			k:=0;
		END_IF
	END_FOR	
			
			(*
			IF en_arch_P THEN
				log_message:=concat(mid(DT_TO_STRING(plc_prg.time_of_st),len(DT_TO_STRING(plc_prg.time_of_st))-2,3),concat(';Измеренный вес, кг:;',concat(REAL_TO_STRING(plc_prg.measured_weight),'$N')));
				point_byte:=ADR(log_message);
				FOR J:=0 TO len(log_message) DO
					buffer_1[k] := point_byte^[J];
					//point_byte:=point_byte+1;
					k:=k+1;
					IF k>=990 THEN
						k:=0;
					END_IF
				END_FOR	
			END_IF
			
			IF en_arch_I THEN
				log_message:=concat(mid(DT_TO_STRING(PLC_PRG.time_of_st),len(DT_TO_STRING(plc_prg.time_of_st))-3,4),concat(';Измеренный вес в процентах, %:;',concat(REAL_TO_STRING(plc_prg.measured_percent),'$N')));
				point_byte:=ADR(log_message);
					FOR J:=0 TO len(log_message) DO
						buffer_1[k] := point_byte^[J];
						//point_byte:=point_byte+1;
						k:=k+1;
						IF k>=990 THEN
							k:=0;
						END_IF
					END_FOR	
				END_IF
			
			IF en_arch_Z THEN
				log_message:=concat(mid(DT_TO_STRING(PLC_PRG.time_of_st),len(DT_TO_STRING(plc_prg.time_of_st))-3,4),concat(';Измеренное напряжение, мВ:;',concat(REAL_TO_STRING(plc_prg.voltage_measurement),'$N')));
				point_byte:=ADR(log_message);
				FOR J:=0 TO len(log_message) DO
					buffer_1[k] := point_byte^[J];
					//point_byte:=point_byte+1;
					k:=k+1;
					IF k>=990 THEN
						k:=0;
					END_IF
				END_FOR	
			END_IF
			*)
	arch_timer(IN:=FALSE);
	
	//IF en_arch_P OR en_arch_I OR en_arch_Z THEN
		IF in_system AND log_write_done AND NOT unmount THEN
		log_write_done:=FALSE;//разрешение на запись
		END_IF
	//END_IF
END_IF	



Archivation();
// /dev/sda1 FLASH
// /dev/mmcblk0p1 SD
IF unmount THEN
	en_arch_P	:=FALSE;
	en_arch_I	:=FALSE;
	en_arch_Z	:=FALSE;
	arch_en:=false;
	um_ton(IN:=TRUE , PT:=T#1S , Q=> , ET=> );
	IF log_write_done AND um_ton.Q THEN
		um_ton(IN:=FALSE);
		sysExecute(sys_command:='umount /dev/mmcblk0p1' );
		unmount:=FALSE;
		//sys3(cmd:= 'umount  /dev/sda1',output_string=> w);
	END_IF
	//sys3(cmd:= 'rm -rf /mnt/ufs/media/sda1',output_string=> w);
	//sys3(cmd:= 'rm -rf /mnt/ufs/media/sda',output_string=> w);
	//sys3(cmd:= 'sync');
	//IF sys3.complete THEN
	
	//END_IF
END_IF
END_ACTION

ACTION Work_with_Flash:
memory_trafo(
	IN:= memory_percent, 
	IN_MIN:=0 , 
	IN_MAX:=100 , 
	OUT_MIN:=358 , 
	OUT_MAX:=1 , 
	OUT=>memory_free_rotate , 
	ERROR=> );
 
rescan_timer(IN:=TRUE , PT:=SEL(in_system,T#5S,T#1M) , Q=> , ET=> );

unmount_F_trig(CLK:=unmount , Q=> );
arch_timer(IN:=arch_en , PT:=DWORD_TO_TIME(Arch_timout*1000) ,Q=> ,ET=> );
IF rescan_timer.Q OR  unmount_F_trig.Q THEN
	may_in_sys:=FALSE;
	scan_flash:=TRUE;
	rescan_timer(in:=FALSE);
END_IF
(*IF scan_flash and not take_info THEN
	reset_in_sys(CLK:=scan_flash , Q=> );
	IF reset_in_sys.Q THEN
		in_system:=FALSE;
		i:=0;
		anti_empty:='';
		FOR i :=0 TO 5 DO
			flash_info[i]:='';
			
		END_FOR
	END_IF
	sys3(cmd:= 'mount', output_string=> w, complete=> );
	IF w<>''THEN
		anti_empty:=w;
	END_IF
	IF find (w,'sda1')<>0  THEN
		in_system:=TRUE;
		trig_to_find_info(CLK:=FALSE);
		//scan_flash:=FALSE;
	END_IF
	IF w='' AND  anti_empty<>'' THEN
		reset_in_sys(CLK:=FALSE);
		scan_flash:=FALSE;
		i:=0;
		
	END_IF
	
END_IF

trig_to_find_info(CLK:=in_system AND NOT scan_flash  , Q=> ); 
IF trig_to_find_info.Q THEN
	take_info:=TRUE;
END_IF*)
// dev/mmcblk0p1 SD
// dev/sda1 FLASH
IF scan_flash THEN 
	//	sys3(cmd:= 'df', output_string=> w, complete=> );
		sys3(cmd:= 'df', output_string=> w, complete=> );
		
		IF find( w, 'dev/mmcblk0p1')<>0 THEN
			may_in_sys:=TRUE;
			FOR i := 0 TO 5 DO
				flash_info[i] :=mid(w,find(w,' '),1);
				
				w:=mid(w,len(w)-find(w,' '),find(w,' '));
				WHILE find(w,' ')=1 DO
					w:=mid(w,len(w)-1,2);
				END_WHILE
			END_FOR
		END_IF
		
		IF w='' AND sys3.complete THEN
			scan_flash:=FALSE;		
		END_IF
		
		IF may_in_sys THEN
			can_arch:=TRUE;
			in_system:=TRUE;
		END_IF
		IF  NOT may_in_sys AND sys3.complete   THEN
			in_system:=FALSE;
			CAN_ARCH:=false;
			
		END_IF
		
		
END_IF

info_trig(CLK:=scan_flash, Q=> );
IF info_trig.Q THEN
	
	IF NOT (flash_info[0]='') THEN
		FOR i:=0 TO 5 DO 
			memory_all:=flash_info[i-3];
			memory_used:=DWORD_TO_WSTRING(STRING_TO_DWORD(flash_info[i-1])/1024);
			memory_all_word:=STRING_TO_DWORD(flash_info[i-1]);
		//	memory_used:=STRING_TO_WSTRING(concat(REAL_TO_STRING((DWORD_TO_REAL(STRING_TO_DWORD(memory_all)-WSTRING_TO_DWORD(memory_used)))/1024),', Мб'));
			IF find (flash_info[i] ,'%')<>0 THEN
				memory_percent:=STRING_TO_REAL(mid(flash_info[i],(len(flash_info[i])-1),1));
				EXIT;
			END_IF
		END_FOR
		IF memory_percent>96 THEN 
			arch_en:=FALSE;
		END_IF
		IF len(memory_all)>6 THEN
			memory_all:=concat(concat(mid(memory_all,(len(memory_all)-7),1),',') , mid ( memory_all, 2, len(memory_all)-6)) ; 
		END_IF
	END_IF	
	
	IF  NOT in_system   THEN
			memory_all_word:=0;
			memory_all:='0,0';
			memory_percent:= 0;
			memory_used:="Flash накопитель отсутствует";
		END_IF
	
		
END_IF



make_log_collection();
END_ACTION

END_PROGRAM

// Device/Application/SearchFile
PROGRAM SearchFile
VAR_INPUT
	temple_name:STRING;//Название файла
	dir:STRING;//Директория для поиска файла (USB/SD, папка)
	file_list:STRING;//Список файлов в файле file_list
	get_list:BOOL; 
END_VAR

VAR_OUTPUT
	list:ARRAY[1..10] OF STRING(255);
	size_list:INT;	
END_VAR

VAR
	req:STRING(255);
	w : STRING;
	sys3 : sysExecute2;
	done:BOOL;
	i:INT;
	pos:INT;
	len_s:int;
END_VAR

done:=FALSE;
size_list:=0;
FOR i:=0 TO 10 DO
	list[i]:='';	
END_FOR
IF get_list THEN//Создаем файл в директории dir - содержащий список файлов в директории dir_list
	
	WHILE(NOT(done))DO
		req:=concat('ls -l ',concat(dir,concat('>',concat(dir,file_list))));
		sys3(cmd:=req,output_string=>w,complete=>done);
	END_WHILE
	
ELSE//поиск
	
	WHILE(NOT(done))DO
		
		req:=concat('ls ',dir);
		sys3(cmd:=req,output_string=>w,complete=>done);
		pos:=find(w,temple_name);
		IF pos<>0 THEN
			pos:=find(w,'$N');
			w:=mid(w,len(w)-1,1);
			IF len(w)>0 THEN
				size_list:=size_list+1;	
				IF size_list<=10 THEN
					list[size_list]:=w;		
				END_IF
			END_IF
		END_IF
		
	END_WHILE	
	
END_IF
(*	
	req:=concat('find ',concat(dir,concat(' -name *',concat(temple_name,'*'))));
	sys3(cmd:=req,output_string=>w,complete=>done);
	w:=mid(w,len(w)-len(ProgramFiles),len(ProgramFiles)+1);

	pos:=find(w,'$N');
	IF pos=len(w) THEN
		w:=mid(w,len(w)-1,1);	
	END_IF
	
	IF len(w)>0 THEN
		size_list:=size_list+1;	
		IF size_list<=10 THEN
			list[size_list]:=w;		
		END_IF
	END_IF
*)

END_PROGRAM

// Device/Application/READ_PROGRAM_FROM_FILE
PROGRAM READ_PROGRAM_FROM_FILE

VAR_INPUT
	name_file_prog:STRING(255):='1.txt';
	begin: BOOL;
END_VAR

VAR_OUTPUT
	PROG_READ:BOOL;
	xError:BOOL;
	FileError:INT;
	Error:INT;(*1-Пустой файл, 2-Файл содержит недопустимый символ переноса строки, 
			3-Некорректное расширение файла (.txt должно быть) либо название файла некорректно,4-зависание функции чтения файла
			5-в файле не хватает данных(точка начала, число зон или другие параметры или нету символа перевода строки в конце файла)*)
END_VAR			

VAR
	init:BOOL;
	ARR_TMPL:ARRAY[1..7] OF STRING(255);
	TMPL_param_N_zon: STRING(255):='Число зон: = ';
	TMPL_param_0 : STRING(255):='Начало низ/верх: = ';
	TMPL_Zakalka_on : STRING(255):='Закалка: = ';
	TMPL_Otpusk_on : STRING(255):='Отпуск: = ';
	TMPL_Rotation : STRING(255):='Вращение: = ';
	TMPL_Spreer : STRING(255):='Спреер преднагрев: = ';
	TMPL_BezSili : STRING(255):='Без силы: = ';
	TMPL_Loxl : STRING(255):='Перемещение охлаждения: = ';
	
	TMPL_param_P_0 : STRING(255):='Начальный нагрев: = ';	
	TMPL_param_t_0 : STRING(255):='Время нач. нагрева: = ';
	TMPL_param_P_L : STRING(255):='Мощность нагрева: = ';
	TMPL_param_L_Zoni : STRING(255):='Длина зоны: = ';
	TMPL_param_V_ind : STRING(255):='Скорость перемещения: = ';
	TMPL_param_t_freeze : STRING(255):='Время конечного охлаждения: = ';
	TMPL_param_R_megdu_zonami : STRING(255):='Расстояние до следующей зоны: = ';

	read_next_line:BOOL;
	Fnd_N_zon, Fnd_0, Fnd_Zakalka_on, Fnd_Otpusk_on, Fnd_Rotation, Fnd_Sreer, Fnd_BezSili, Fnd_Loxl :BOOL;//Загаловок
	Fnd_Params : ARRAY[1..10,1..7] OF BOOL;
	Fnd_zones : ARRAY[1..10] OF BOOL;
	Zona:INT:=1;
	ZONA_READ:BOOL;
	END_OF_FILE:BOOL;
	
	check_name_file:BOOL;
	pos: INT;
	end_line_point: INT;
	position:UDINT;
	buf_pos:UDINT;
	value_test:INT;
	FND_NEXT_PARAM: BOOL;
	
	Props_open: FILE.Open;
	Props_read: FILE.Read;
	str_buf: STRING(255);

	props_set_pos: FILE.SetPos;
	get_size: FILE.GetSize;
	size_file: UDINT;
	read_state: INT:=0;
	
	count: INT;
	cnt_freeze:INT;
	Place_Freezes:INT; //Завис при выполнение фу-ии :1- get_size,2- Props_open,3- Props_read,4- props_set_pos,5- 90 props_close,6- 100 props_close
	err_count: INT;
	props_close: FILE.Close;
	
	i:INT:=1;(*используются в Analyz_str*)
	buf_i: INT;
	buf_j:INT;
	tmp:INT;
	tmp_bool:INT;
	
	ptr_byte: POINTER TO BYTE;
	symbol_code: BYTE;
	j:INT;
	FND_SYMBOL:BOOL;
END_VAR

IF begin THEN
	
	IF NOT(init) THEN
		init:=TRUE;
		ARR_TMPL[1]:=TMPL_param_P_0;
		ARR_TMPL[2]:=TMPL_param_t_0;
		ARR_TMPL[3]:=TMPL_param_P_L;
		ARR_TMPL[4]:=TMPL_param_L_Zoni;
		ARR_TMPL[5]:=TMPL_param_V_ind;
		ARR_TMPL[6]:=TMPL_param_t_freeze;
		ARR_TMPL[7]:=TMPL_param_R_megdu_zonami;
	END_IF

IF NOT(check_name_file) THEN
	pos:=find(name_file_prog,'.txt');
	IF 	pos<>0 AND len(name_file_prog)>4 THEN
		pos:=find(name_file_prog,'$N');
		IF pos=0 THEN
			check_name_file:=TRUE;
			xError:=FALSE;
			Error:=0;
		ELSE
			check_name_file:=FALSE;
			Error:=2;//Файл содержит недопустимый символ переноса строки
			xError:=TRUE;
		END_IF
	ELSE
		check_name_file:=FALSE;
		Error:=3;//Некорректное расширение файла (.txt должно быть) либо название файла некорректно
		xError:=TRUE;
	END_IF
END_IF
			
IF check_name_file THEN
	CASE read_state OF
	0:	get_size(
			xExecute:= TRUE, 
			xDone=> , 
			xBusy=> , 
			xError=> xError, 
			sFileName:=concat(ProgramFiles,name_file_prog) , 
			eError=> FileError, 
			szSize=>size_file);
		Place_Freezes:=1;	
		cnt_freeze:=cnt_freeze+1;	
		IF get_size.xDone THEN
			cnt_freeze:=0;
			IF size_file = 0 THEN
				read_state := 89;
			END_IF
			read_state:=1;
			get_size(xExecute:= FALSE);
		END_IF
		
		IF get_size.xError THEN
			cnt_freeze:=0;
			read_state:=0;
			err_count:=err_count+1;
			IF err_count>=3 THEN
				err_count:=0;
				read_state:=90;
			END_IF
		END_IF

		IF cnt_freeze>10 THEN
			read_state:=88;//Зависание функции чтения
			cnt_freeze:=0;
		END_IF	
		
		1:
		Props_open(
			xExecute:=TRUE , 
			xDone=> , 
			xBusy=> , 
			xError=> xError, 
			sFileName:=concat(ProgramFiles,name_file_prog) , 
			eFileMode:=FILE.MODE.MREAD , 
			xExclusive:= , 
			eError=>FileError , 
			hFile=>);
		Place_Freezes:=2;	
		cnt_freeze:=cnt_freeze+1;	
		IF Props_open.xDone THEN
			cnt_freeze:=0;
			position:=0;
			read_next_line:=TRUE;
			read_state:=2;
			ClearBuf(p:=ADR(str_buf));
			
			Fnd_N_zon:=FALSE;
			Fnd_0:=FALSE;
			Fnd_Zakalka_on:=FALSE;
			Fnd_Otpusk_on:=FALSE;
			Fnd_Rotation:=FALSE;
			Fnd_Sreer:=FALSE;
			Fnd_BezSili:=FALSE; 
			Fnd_Loxl:=FALSE;
			
			(*обнуление текущей программы закалки*)
			chislo_zon := 0;
			ZAKALKA.zakalka_nachalo := 0;
			FOR Zona:=1 TO 10 DO
				P_nachaln_nagrev[Zona]:=1;
				t_nachaln_nagrev[Zona]:=0;
				P_nagrev[Zona]:=1;
				L_peremeshenia[Zona]:=0;
				V_peremeshenia[Zona]:=0;
				t_freeze[Zona]:=0;
				L_to_next_zone[Zona]:=0;
				
				Fnd_zones[Zona]:=FALSE;
				FOR i:=1 TO 7 DO 
					Fnd_Params[Zona,i]:=FALSE;
				END_FOR
			END_FOR
			Zona:=1;
			i:=1;
			PROG_READ:=FALSE;
		END_IF
		
		IF cnt_freeze>10 THEN
			read_state:=88;//Зависание функции чтения
			cnt_freeze:=0;
		END_IF	
		
		2:Props_read(
				xExecute:=TRUE , 
				xAbort:= , 
				udiTimeOut:= , 
				xDone=> , 
				xBusy=> , 
				xError=> xError, 
				xAborted=> , 
				hFile:=Props_open.hFile, 
				pBuffer:=ADR(str_buf) , 
				szBuffer:=SEL(read_next_line,0,SIZEOF(str_buf)-1) , 
				eError=> FileError, 
				szSize=> );
			Place_Freezes:=3;	
			cnt_freeze:=cnt_freeze+1;
	
			
			IF Props_read.xDone THEN
				cnt_freeze:=0;
				buf_pos:=position;

				Analyz_str();
				
				IF FND_NEXT_PARAM THEN
					read_next_line:=FALSE;
					read_state:=2;
				ELSE
					read_next_line:=TRUE;
					read_state:=3;
					IF position=buf_pos THEN
						Find_Symbol();//Ищет позицию первого символ кирилицы или цифры - j-индекс первого символа
						IF FND_SYMBOL THEN
							position:=position+j;
						ELSE
							position:=position+255;
						END_IF
						IF (position)>=size_file THEN
							read_state:=90;//был прочитан конец файла
						END_IF
					END_IF
				END_IF
				
				IF PROG_READ THEN
					read_state:=100;
				END_IF
				
				IF END_OF_FILE OR NOT(Fnd_0) OR NOT(Fnd_N_zon) THEN
					read_state:=90;
					Error:=5;
				END_IF
				
				Props_read(xExecute:=FALSE);
			END_IF
			
			IF Props_read.xError THEN
				cnt_freeze:=0;
				err_count:=err_count+1;
				IF err_count>=3 THEN
					err_count:=0;
					read_state:=90;
				END_IF
			END_IF
			
			IF cnt_freeze>10 THEN
				read_state:=88;//Зависание функции чтения
				cnt_freeze:=0;
			END_IF
			
		3:props_set_pos(
			xExecute:= TRUE, 
			xDone=> , 
			xBusy=> , 
			xError=> xError, 
			hFile:=Props_open.hFile , 
			udiPos:=position , 
			eError=> FileError);
		Place_Freezes:=4;	
		cnt_freeze:=cnt_freeze+1;
	
		IF props_set_pos.xDone THEN
			cnt_freeze:=0;
			read_state:=2;
			ClearBuf(p:=ADR(str_buf));
			props_set_pos(xExecute:= false);
		END_IF
		
		IF props_set_pos.xError THEN
			cnt_freeze:=0;
			read_state:=3;
			err_count:=err_count+1;
				IF err_count>=3 THEN
					err_count:=0;
					read_state:=90;
				END_IF
		END_IF
		
		IF cnt_freeze>10 THEN
			read_state:=88;//Зависание функции чтения
			cnt_freeze:=0;
		END_IF
		
	88://Зависание функции чтения файла
	read_state:=0;
	check_name_file:=FALSE;
	begin:=FALSE;
	Error:=4;//Зависание функции чтения файла
	xError:=TRUE;
				
	89://File Size=0
	read_state:=0;
	check_name_file:=FALSE;
	begin:=FALSE;
	Error:=1;//Пустой файл
	xError:=TRUE;
	
	90:
	props_close(
	xExecute:=TRUE , 
	xDone=> , 
	xBusy=> , 
	xError=> xError, 
	hFile:=Props_open.hFile , 
	eError=> FileError);
	Place_Freezes:=5;
	cnt_freeze:=cnt_freeze+1;
	
	IF props_close.xDone THEN
		cnt_freeze:=0;
		begin:=FALSE;
		Zona:=1;
		i:=1;
		check_name_file:=FALSE;
		read_state:=0;
		PROG_READ:=FALSE;
		
		Props_open(xExecute:=FALSE);
		props_close(xExecute:=FALSE);
	END_IF
	
	IF props_close.xError THEN
		cnt_freeze:=0;
		begin:=FALSE;
		Zona:=1;
		i:=1;
		check_name_file:=FALSE;
		read_state:=0;
		PROG_READ:=FALSE;
		
		Props_open(xExecute:=FALSE);
		props_close(xExecute:=FALSE);
	END_IF
	
		IF cnt_freeze>10 THEN
			read_state:=88;//Зависание функции чтения
			cnt_freeze:=0;
		END_IF		
	100:
	props_close(
	xExecute:=TRUE , 
	xDone=> , 
	xBusy=> , 
	xError=> xError, 
	hFile:=Props_open.hFile , 
	eError=> FileError);
	Place_Freezes:=6;
	cnt_freeze:=cnt_freeze+1;

	IF props_close.xDone THEN
		cnt_freeze:=0;
		begin:=FALSE;
		Zona:=1;
		i:=1;
		check_name_file:=FALSE;
		read_state:=0;
		
		Props_open(xExecute:=FALSE);
		props_close(xExecute:=FALSE);
	END_IF
	
	IF props_close.xError THEN
		cnt_freeze:=0;
		begin:=FALSE;
		Zona:=1;
		i:=1;
		check_name_file:=FALSE;
		read_state:=0;
		
		Props_open(xExecute:=FALSE);
		props_close(xExecute:=FALSE);
	END_IF
	
		IF cnt_freeze>10 THEN
			read_state:=88;//Зависание функции чтения
			cnt_freeze:=0;
		END_IF		
		
	END_CASE	
END_IF

END_IF

ACTION Analyz_str:
//////////////////////////////////////////////////Считывание Заголовка/////////////////////////////////////////////////////////////////
//Число зон TMPL_param_N_zon || Fnd_N_zon
IF NOT(Fnd_N_zon) THEN
	RD_param(temple_param:=TMPL_param_N_zon, str_buf:=str_buf,value=>chislo_zon,FND_PARAM=>Fnd_N_zon,index=>end_line_point);
	IF Fnd_N_zon THEN
		str_buf:=mid(str_buf,len(str_buf)-end_line_point,end_line_point+1);//вырезаем из строки прочитанный параметр
		position:=position+end_line_point;//переносим указатель на следующий параметр
	END_IF
END_IF	

//Начало TMPL_param_0 || Fnd_0
IF NOT(Fnd_0) THEN
	RD_param(temple_param:=TMPL_param_0, str_buf:=str_buf, value=>ZAKALKA.zakalka_nachalo, FND_PARAM=>Fnd_0, index=>end_line_point);
	IF Fnd_0 THEN
		str_buf:=mid(str_buf,len(str_buf)-end_line_point,end_line_point+1);
		position:=position+end_line_point;
	END_IF
END_IF

//Закалка TMPL_Zakalka_on || Fnd_Zakalka_on -> ZAKALKA.Zakalka_on
IF NOT(Fnd_Zakalka_on) THEN
	RD_param(temple_param:=TMPL_Zakalka_on, str_buf:=str_buf, value=>tmp_bool, FND_PARAM=>Fnd_Zakalka_on, index=>end_line_point);
	ZAKALKA.Zakalka_on:=SEL(tmp_bool=1,FALSE,TRUE);
	IF Fnd_Zakalka_on THEN
		str_buf:=mid(str_buf,len(str_buf)-end_line_point,end_line_point+1);
		position:=position+end_line_point;
	END_IF
END_IF					

//Отпуск TMPL_Otpusk_on || Fnd_Otpusk_on -> ZAKALKA.Otpusk_on
IF NOT(Fnd_Otpusk_on) THEN
	RD_param(temple_param:=TMPL_Otpusk_on, str_buf:=str_buf, value=>tmp_bool, FND_PARAM=>Fnd_Otpusk_on, index=>end_line_point);
	ZAKALKA.Otpusk_on:=SEL(tmp_bool=1,FALSE,TRUE);
	IF Fnd_Otpusk_on THEN
		str_buf:=mid(str_buf,len(str_buf)-end_line_point,end_line_point+1);
		position:=position+end_line_point;
	END_IF
END_IF

//Вращение TMPL_Rotation || Fnd_Rotation -> ZAKALKA.rotation_on
IF NOT(Fnd_Rotation) THEN
	RD_param(temple_param:=TMPL_Rotation, str_buf:=str_buf, value=>tmp_bool, FND_PARAM=>Fnd_Rotation, index=>end_line_point);
	ZAKALKA.rotation_on:=SEL(tmp_bool=1,FALSE,TRUE);
	IF Fnd_Rotation THEN
		str_buf:=mid(str_buf,len(str_buf)-end_line_point,end_line_point+1);
		position:=position+end_line_point;
	END_IF
END_IF	

//Спреер преднагрев TMPL_Spreer || Fnd_Sreer -> ZAKALKA.spreer_prednagrev
IF NOT(Fnd_Sreer) THEN
	RD_param(temple_param:=TMPL_Spreer, str_buf:=str_buf, value=>tmp_bool, FND_PARAM=>Fnd_Sreer, index=>end_line_point);
	ZAKALKA.spreer_prednagrev:=SEL(tmp_bool=1,FALSE,TRUE);
	IF Fnd_Sreer THEN
		str_buf:=mid(str_buf,len(str_buf)-end_line_point,end_line_point+1);
		position:=position+end_line_point;
	END_IF
END_IF

//Без силы TMPL_BezSili || Fnd_BezSili -> ZAKALKA.diagnostik
IF NOT(Fnd_BezSili) THEN
	RD_param(temple_param:=TMPL_BezSili, str_buf:=str_buf, value=>tmp_bool, FND_PARAM=>Fnd_BezSili, index=>end_line_point);
	ZAKALKA.diagnostik:=SEL(tmp_bool=1,FALSE,TRUE);
	IF Fnd_BezSili THEN
		str_buf:=mid(str_buf,len(str_buf)-end_line_point,end_line_point+1);
		position:=position+end_line_point;
	END_IF
END_IF		

//TMPL_param_R_oxl -> Fnd_R -> L_peremesh_ohl GVL
IF NOT(Fnd_Loxl) THEN
	RD_param(fnd_end:=FALSE,temple_param:=TMPL_Loxl, str_buf:=str_buf, value=>L_peremesh_ohl, FND_PARAM=>Fnd_Loxl, index=>end_line_point);
	IF Fnd_Loxl THEN
		str_buf:=mid(str_buf,len(str_buf)-end_line_point,end_line_point+1);
		position:=position+end_line_point;
	END_IF 
END_IF

///////////////////////////////////////////////Считывание ЗОНЫ//////////////////////////////////////////////////////////////////////
//Мощность на преднагреве TMPL_param_P_0 || Fnd_P_0
IF NOT(Fnd_Params[Zona,1]) THEN
	RD_param(fnd_end:=FALSE,temple_param:=TMPL_param_P_0, str_buf:=str_buf, value=>P_nachaln_nagrev[Zona], FND_PARAM=>Fnd_Params[Zona,1], index=>end_line_point);
	IF Fnd_Params[Zona,1] THEN
		str_buf:=mid(str_buf,len(str_buf)-end_line_point,end_line_point+1);//Резать не всю строку а убирать из нее прочитанный параметр
		position:=position+end_line_point;//Надо реализовать функцию которая вырезает из строки отрезок по индексам [1..5] например
	END_IF
END_IF

//время на преднагреве TMPL_param_t_0 || Fnd_t_0
IF NOT(Fnd_Params[Zona,2]) THEN
	RD_param(fnd_end:=FALSE,temple_param:=TMPL_param_t_0, str_buf:=str_buf, value=>t_nachaln_nagrev[Zona], FND_PARAM=>Fnd_Params[Zona,2], index=>end_line_point);
	IF Fnd_Params[Zona,2] THEN
		str_buf:=mid(str_buf,len(str_buf)-end_line_point,end_line_point+1);
		position:=position+end_line_point;
	END_IF	
END_IF

//Мощность в движении TMPL_param_P_L || Fnd_P_L
IF NOT(Fnd_Params[Zona,3]) THEN
	RD_param(fnd_end:=FALSE,temple_param:=TMPL_param_P_L, str_buf:=str_buf, value=>P_nagrev[Zona], FND_PARAM=>Fnd_Params[Zona,3], index=>end_line_point);
	IF Fnd_Params[Zona,3] THEN
		str_buf:=mid(str_buf,len(str_buf)-end_line_point,end_line_point+1);
		position:=position+end_line_point;
	END_IF	
END_IF

//Длина зоны TMPL_param_L_Zoni || Fnd_L_Z
IF NOT(Fnd_Params[Zona,4]) THEN
	RD_param(fnd_end:=FALSE,temple_param:=TMPL_param_L_Zoni, str_buf:=str_buf, value=>L_peremeshenia[Zona], FND_PARAM=>Fnd_Params[Zona,4], index=>end_line_point);
	IF Fnd_Params[Zona,4] THEN
		str_buf:=mid(str_buf,len(str_buf)-end_line_point,end_line_point+1);
		position:=position+end_line_point;
	END_IF	
END_IF

// скорость индуктора TMPL_param_V_ind || Fnd_V_ind
IF NOT(Fnd_Params[Zona,5]) THEN
	RD_param(fnd_end:=FALSE,temple_param:=TMPL_param_V_ind, str_buf:=str_buf, value=>V_peremeshenia[Zona], FND_PARAM=>Fnd_Params[Zona,5], index=>end_line_point);
	IF Fnd_Params[Zona,5] THEN
		str_buf:=mid(str_buf,len(str_buf)-end_line_point,end_line_point+1);
		position:=position+end_line_point;
	END_IF	
END_IF

//TMPL_param_t_freeze || Fnd_Toxl
IF NOT(Fnd_Params[Zona,6]) THEN
	RD_param(fnd_end:=FALSE,temple_param:=TMPL_param_t_freeze, str_buf:=str_buf, value=>t_freeze[Zona], FND_PARAM=>Fnd_Params[Zona,6], index=>end_line_point);
	IF Fnd_Params[Zona,6] THEN
		str_buf:=mid(str_buf,len(str_buf)-end_line_point,end_line_point+1);
		position:=position+end_line_point;
	END_IF	
END_IF

//TMPL_param_R_megdu_zonami || Fnd_R
IF NOT(Fnd_Params[Zona,7]) THEN
	RD_param(fnd_end:=FALSE,temple_param:=TMPL_param_R_megdu_zonami, str_buf:=str_buf, value=>L_to_next_zone[Zona], FND_PARAM=>Fnd_Params[Zona,7], index=>end_line_point);
	IF Fnd_Params[Zona,7] THEN
		str_buf:=mid(str_buf,len(str_buf)-end_line_point,end_line_point+1);
		position:=position+end_line_point;
	END_IF 
END_IF

ZONA_READ:=Fnd_Params[Zona,1] AND Fnd_Params[Zona,2] AND Fnd_Params[Zona,3] AND Fnd_Params[Zona,4] AND Fnd_Params[Zona,5] AND Fnd_Params[Zona,6] AND Fnd_Params[Zona,7];

IF ZONA_READ THEN
	IF Zona<chislo_zon THEN
		Fnd_zones[Zona]:=TRUE;
		Zona:=Zona+1;
		ZONA_READ:=FALSE;
	ELSE
		PROG_READ:=TRUE;
		read_state:=100;
	END_IF
END_IF
				

buf_i:=-1;
FOR i:=1 TO 10 DO
	IF NOT(Fnd_zones[i]) THEN
		buf_i:=i;
		EXIT;
	END_IF
END_FOR

buf_j:=-1;
IF Zona <> chislo_zon THEN
	FOR i:=1 TO 7 DO
		IF NOT(Fnd_Params[buf_i,i]) THEN
			buf_j:=i;
			EXIT;
		END_IF
	END_FOR
ELSE
	FOR i:=1 TO 7 DO
		IF NOT(Fnd_Params[buf_i,i]) THEN
			buf_j:=i;
			EXIT;
		END_IF
	END_FOR
	
		
END_IF

IF buf_j>0 THEN
	RD_param(fnd_end:=TRUE, position:=position, size_file:=size_file, temple_param:=ARR_TMPL[buf_j], str_buf:=str_buf, value=>value_test, FND_PARAM=>FND_NEXT_PARAM, index=>end_line_point,END_OF_FILE=>END_OF_FILE);//проверка на конец файла
	IF END_OF_FILE THEN
		CASE buf_j OF 
			1:P_nachaln_nagrev[Zona]:=value_test;
			2:t_nachaln_nagrev[Zona]:=value_test;
			3:P_nagrev[Zona]:=value_test;
			4:L_peremeshenia[Zona]:=value_test;
			5:V_peremeshenia[Zona]:=value_test;
			6:t_freeze[Zona]:=value_test;
			7:L_to_next_zone[Zona]:=value_test;
		END_CASE
	END_IF
END_IF
END_ACTION

ACTION Find_Symbol:
FND_SYMBOL:=FALSE;
ptr_byte:=ADR(str_buf);

FOR j:=0 TO 255 DO
	symbol_code:=ptr_byte[j];
	IF (symbol_code>=48 AND symbol_code<=57) OR symbol_code=58 OR symbol_code=61 OR symbol_code=91 OR symbol_code=93 THEN//нашли цифры или ':' или '=' или '[' или ']'
		FND_SYMBOL:=TRUE;
		EXIT;
	END_IF
	IF symbol_code>=192 AND symbol_code<=255 THEN//нашли символ из кирилицы
		FND_SYMBOL:=TRUE;
		EXIT;
	END_IF
END_FOR
END_ACTION

END_PROGRAM

// Device/Application/ClearBuf
PROGRAM ClearBuf
VAR_INPUT
	p:POINTER TO BYTE;
	i:INT;
END_VAR

VAR
END_VAR

FOR i:=0 TO 255 DO
	p[i]:=0;
END_FOR
RETURN;

END_PROGRAM

// Device/Application/RD_param
PROGRAM RD_param 

VAR_INPUT
	temple_param:STRING(255);//Название параметра
	str_buf:STRING(255);//строка из файла .ini
	position:UDINT;//позиция чтения файла
	size_file:UDINT;//размер файла
	fnd_end:BOOL:=false;
END_VAR

VAR_OUTPUT
	value:INT;
	FND_PARAM:BOOL;
	FND_DIGITS:BOOL;
	index:INT;//указывает на конец строки в которой был найден параметр
	END_OF_FILE:BOOL;
END_VAR

VAR
	i_digits,pos,i: INT;
	
	ptr_str_buf:POINTER TO BYTE;
	ptr_str_value:POINTER TO BYTE;
	str_value : STRING(255);
	byte_s : BYTE;
END_VAR

//ASCII(DEC) 48 49 50 51 52 53 54 55 56 57
//SYMBOL      0  1  2  3  4  5  6  7  8  9
value:=0;
FND_PARAM:=FALSE;
i_digits:=0;
IF NOT(fnd_end) THEN
	END_OF_FILE:=FALSE;
	pos:=find(str_buf,temple_param);
	IF pos<>0 THEN
	ptr_str_buf:=ADR(str_buf);
	ptr_str_value:=ADR(str_value);
	i:=pos+len(temple_param)-1;

	WHILE (i <= LEN(str_buf)) AND NOT(FND_PARAM) DO
		byte_s:=ptr_str_buf[i];//индексация от 0 до 255
		IF (byte_s>=48 AND byte_s<=57) OR  byte_s=10 OR byte_s=13 OR byte_s=0 THEN
			ptr_str_value[i_digits]:=byte_s;
			i_digits:=i_digits+1;
			IF byte_s=10 OR byte_s=0  THEN
				FND_PARAM:=TRUE;
				value:=STRING_TO_INT(str_value);
				index:=i+1;
			END_IF
		END_IF
		i:=i+1;
	END_WHILE
	END_IF
ELSE
	pos:=find(str_buf,temple_param);
	IF pos<>0 THEN
	ptr_str_buf:=ADR(str_buf);
	ptr_str_value:=ADR(str_value);
	i:=pos+len(temple_param)-1;
	WHILE (i <= LEN(str_buf)) AND NOT(FND_PARAM) DO
		byte_s:=ptr_str_buf[i];//индексация от 0 до 255
		IF (byte_s>=48 AND byte_s<=57) OR  byte_s=10 OR byte_s=13 OR byte_s=0 THEN
			ptr_str_value[i_digits]:=byte_s;
			i_digits:=i_digits+1;
			IF byte_s=10 OR byte_s=0 THEN//найден символ перевода на следующую строку
				FND_PARAM:=TRUE;
				value:=STRING_TO_INT(str_value);
				index:=i+1;
			END_IF
		END_IF
		
		i:=i+1;
		IF position+i>=size_file THEN
			value:=STRING_TO_INT(str_value);
			END_OF_FILE:=TRUE;
		END_IF
	END_WHILE
	END_IF
END_IF

END_PROGRAM

// Device/Application/WRITE_PROGRAM_FILE_ON_SD
PROGRAM WRITE_PROGRAM_FILE_ON_SD

VAR_INPUT
	name_file:STRING(255);
	wr:BOOL;
END_VAR

VAR_OUTPUT
	xError : BOOL;
	FileError : INT;
	StrError : STRING;
	err_func : INT;
	freeze:BOOL;	
END_VAR

VAR
	TMPL_title: STRING(255):='[Программа]';
	TMPL_param_N_zon: STRING(255):='Число зон: = ';
	TMPL_param_0 : STRING(255):='Начало низ/верх: = ';
	
	TMPL_Zakalka_on : STRING(255):='Закалка: = ';
	TMPL_Otpusk_on : STRING(255):='Отпуск: = ';
	TMPL_Rotation : STRING(255):='Вращение: = ';
	TMPL_Spreer : STRING(255):='Спреер преднагрев: = ';
	TMPL_BezSili : STRING(255):='Без силы: = ';
	TMPL_Loxl : STRING(255):='Перемещение охлаждения: = ';

	TMPL_param_P_0 : STRING(255):='Начальный нагрев: = ';	
	TMPL_param_t_0 : STRING(255):='Время нач. нагрева: = ';
	TMPL_param_P_L : STRING(255):='Мощность нагрева: = ';
	TMPL_param_L_Zoni : STRING(255):='Длина зоны: = ';
	TMPL_param_V_ind : STRING(255):='Скорость перемещения: = ';
	TMPL_param_t_freeze : STRING(255):='Время конечного охлаждения: = ';
	TMPL_param_R_megdu_zonami : STRING(255):='Расстояние до следующей зоны: = ';
	TMPL_param_R_oxl : STRING(255):='Перемещение охлаждения: = '; //L_peremesh_ohl GVL
	TEMP 				: STRING(255);
	i_zona				: INT;
	position			: UDINT;
	
	size_file			: UDINT;
	state_write 		: BYTE:=0;
	open_file			: FILE.Open;
	write_to_file		: FILE.Write;
	close_file			: FILE.Close;
	set_pos				: FILE.SetPos;
	get_size			: FILE.GetSize;
	
	err_count			: BYTE:=0;
	cnt_freeze			: BYTE;
	FileExist : BOOL;
END_VAR

IF wr THEN
	freeze:=FALSE;
	CASE state_write OF
		0:
		IF NOT(find(name_file,'.txt')<>0) THEN
			name_file:=concat(name_file,'.txt');
		END_IF	
		get_size(
			xExecute:= TRUE, 
			xDone=> , 
			xBusy=> , 
			xError=> xError, 
			sFileName:=concat(ProgramFiles, name_file) , 
			eError=> FileError, 
			szSize=> size_file);
			
		cnt_freeze:=cnt_freeze+1;
		IF cnt_freeze>100 THEN
			cnt_freeze:=0;
			state_write:=6;//Зависание функкции записи
		END_IF
		
		IF get_size.xDone THEN
			get_size(xExecute:= FALSE);
			cnt_freeze:=0;
			err_func:=0;
			state_write:=1;
			FileExist:=TRUE;
		ELSIF get_size.xError AND get_size.eError=file.ERROR.NOT_EXIST THEN
			state_write:=1;
			FileExist:=FALSE;
		ELSIF get_size.xError THEN
			FileExist:=FALSE;
			err_count:=err_count+1;
			IF err_count>=3 THEN
				err_count:=0;
				state_write:=5;//ошибочное завершение функции записи на этапе получения размера файла
				err_func := 1;
			END_IF			
		END_IF

		
		1:
		open_file(
		xExecute:=TRUE , 
		xDone=> , 
		xBusy=> , 
		xError=> xError, 
		sFileName:=concat(ProgramFiles,name_file), 
		eFileMode:=file.MODE.MWRITE, 
		xExclusive:=, 
		eError=> FileError, 
		hFile=> );
		
		cnt_freeze:=cnt_freeze+1;
		IF cnt_freeze>100 THEN
			cnt_freeze:=0;
			state_write:=6;//Зависание функкции записи
		END_IF			
		IF open_file.xDone THEN
			position:=0;
			cnt_freeze:=0;
			err_func:=0;
			state_write:=2;
			TEMP:='';
			TEMP:=concat(TMPL_title,'$R$N');//Подключили заголовок
			TEMP:=concat(TEMP,concat(concat(TMPL_param_N_zon,INT_TO_STRING(chislo_zon)),'$R$N'));//Подключили число зон
			TEMP:=concat(TEMP,concat(concat(TMPL_param_0,INT_TO_STRING(ZAKALKA.zakalka_nachalo)),'$R$N'));//Подключили точку начало
			TEMP:=concat(TEMP,concat(concat(TMPL_Zakalka_on,INT_TO_STRING(SEL(ZAKALKA.Zakalka_on,0,1))),'$R$N'));//Закалка
			TEMP:=concat(TEMP,concat(concat(TMPL_Otpusk_on,INT_TO_STRING(SEL(ZAKALKA.Otpusk_on,0,1))),'$R$N'));//Отпуск
			TEMP:=concat(TEMP,concat(concat(TMPL_Rotation,INT_TO_STRING(SEL(ZAKALKA.rotation_on,0,1))),'$R$N'));//Вращение
			TEMP:=concat(TEMP,concat(concat(TMPL_Spreer,INT_TO_STRING(SEL(ZAKALKA.spreer_prednagrev,0,1))),'$R$N'));//Спреер преднагрев
			TEMP:=concat(TEMP,concat(concat(TMPL_BezSili,INT_TO_STRING(SEL(ZAKALKA.diagnostik,0,1))),'$R$N'));//Без силы
			TEMP:=concat(TEMP,concat(concat(TMPL_Loxl,WORD_TO_STRING(L_peremesh_ohl)),'$R$N'));//Перемещение охлаждения
			TEMP:=concat(TEMP,'$R$N');//конец заголовка
			i_zona:=1;
		END_IF
		
		IF open_file.xError THEN
			open_file(xExecute:=FALSE);
			err_count:=err_count+1;
			IF err_count>=3 THEN
				err_func := 2;
				err_count:=0;
				state_write:=5;//ошибочное завершение функции записи на этапе открытия файла
			END_IF
		END_IF	
		
		2:
		write_to_file(
			xExecute:=TRUE , 
			xAbort:= , 
			udiTimeOut:= , 
			xDone=> , 
			xBusy=> , 
			xError=> xError, 
			xAborted=> , 
			hFile:=open_file.hFile , 
			pBuffer:= ADR(TEMP), 
			szSize:= len(TEMP), 
			eError=> FileError);
			
		cnt_freeze:=cnt_freeze+1;
		IF cnt_freeze>100 THEN
			cnt_freeze:=0;
			state_write:=6;//Зависание функкции записи
		END_IF	
 	
		IF write_to_file.xDone  THEN
			cnt_freeze:=0;
			err_func:=0;
			write_to_file(xExecute:= FALSE);
			state_write:=3;
			position:=position+len(TEMP);
		END_IF
		
		IF write_to_file.xError THEN
			err_count:=err_count+1;
			IF err_count>=3 THEN
				err_func:=3;
				err_count:=0;
				state_write:=5;
			END_IF
		END_IF
			
		3:
		set_pos(
			xExecute:= TRUE, 
			xDone=> , 
			xBusy=> , 
			xError=> xError, 
			hFile:=open_file.hFile , 
			udiPos:= position, 	
			eError=>FileError);
			
		cnt_freeze:=cnt_freeze+1;
		IF cnt_freeze>100 THEN
			cnt_freeze:=0;
			state_write:=6;
		END_IF	
			
		IF set_pos.xDone THEN
			cnt_freeze:=0;
			err_func:=0;
			set_pos(xExecute:= FALSE); 
			IF i_zona>chislo_zon THEN
				state_write:=4;//программа записанна полностью
			ELSE
				TEMP:='';
				//Подключаем параметры одной зоны
				TEMP:=concat(concat('[Зона ',INT_TO_STRING(i_zona)),']$R$N');//Заголовок зоны
				TEMP:=concat(TEMP,concat(concat(TMPL_param_P_0,INT_TO_STRING(P_nachaln_nagrev[i_zona])),'$R$N'));
				TEMP:=concat(TEMP,concat(concat(TMPL_param_t_0,INT_TO_STRING(t_nachaln_nagrev[i_zona])),'$R$N'));
				TEMP:=concat(TEMP,concat(concat(TMPL_param_P_L,INT_TO_STRING(P_nagrev[i_zona])),'$R$N'));
				TEMP:=concat(TEMP,concat(concat(TMPL_param_L_Zoni,INT_TO_STRING(L_peremeshenia[i_zona])),'$R$N'));
				TEMP:=concat(TEMP,concat(concat(TMPL_param_V_ind,INT_TO_STRING(V_peremeshenia[i_zona])),'$R$N'));
				TEMP:=concat(TEMP,concat(concat(TMPL_param_t_freeze,INT_TO_STRING(t_freeze[i_zona])),'$R$N'));
				TEMP:=concat(TEMP,concat(concat(TMPL_param_R_megdu_zonami,INT_TO_STRING(L_to_next_zone[i_zona])),'$R$N'));//Текущей или следующей зоны?
				
				IF i_zona<>chislo_zon THEN
					TEMP:=concat(TEMP,'$R$N');//конец заголовка
				END_IF
				i_zona:=i_zona+1;
				state_write:=2;
				
			END_IF
		END_IF
		
		IF set_pos.xError THEN	
			err_count:=err_count+1;
			IF err_count>=3 THEN
				err_func:=4;
				err_count:=0;
				state_write:=5;
			END_IF
		END_IF
		
		4://Успешное завершение записи программы
		close_file(
			xExecute:=TRUE , 
			xDone=> , 
			xBusy=> , 
			xError=> xError, 
			hFile:=open_file.hFile , 
			eError=> FileError);
			
		cnt_freeze:=cnt_freeze+1;
		IF cnt_freeze>100 THEN
			cnt_freeze:=0;
			state_write:=6;//Зависание функкции записи
		END_IF		
		
		IF close_file.xDone THEN
			cnt_freeze:=0;
			open_file(xexecute:=FALSE);
			close_file(xexecute:=FALSE);
			wr:=FALSE;
			state_write:=0;	
		END_IF
		
		IF close_file.xError THEN
			open_file(xexecute:=FALSE);
			close_file(xexecute:=FALSE);
			err_count:=err_count+1;
			IF err_count>=10 THEN
				err_func:=5;
				err_count:=0;
				state_write:=0;
				open_file(xexecute:=FALSE);
				close_file(xexecute:=FALSE);
				wr:=false;
			END_IF
		END_IF
		
		5://Pавершение записи программы с ошибкой
		close_file(
			xExecute:=TRUE , 
			xDone=> , 
			xBusy=> , 
			xError=> xError, 
			hFile:=open_file.hFile , 
			eError=> FileError);
			
		cnt_freeze:=cnt_freeze+1;
		IF cnt_freeze>100 THEN
			cnt_freeze:=0;
			state_write:=6;//Зависание функкции записи
		END_IF
		
		IF close_file.xDone THEN
			cnt_freeze:=0;
			cnt_freeze:=0;
			open_file(xexecute:=FALSE);
			close_file(xexecute:=FALSE);
			wr:=FALSE;
			state_write:=0;	
		END_IF
		
		IF close_file.xError THEN
			cnt_freeze:=0;
			err_func:=6;
			open_file(xexecute:=FALSE);
			close_file(xexecute:=FALSE);
			err_count:=err_count+1;
			IF err_count>=10 THEN
				err_count:=0;
				state_write:=0;
				open_file(xexecute:=FALSE);
				close_file(xexecute:=FALSE);
				wr:=FALSE;
			END_IF
		END_IF
		6://Обработка зависания функции
		cnt_freeze:=0;
		freeze:=TRUE;
		state_write:=0;
		wr:=FALSE;
		open_file(xexecute:=FALSE);
		write_to_file(xexecute:=FALSE);
		get_size(xexecute:=FALSE);
		set_pos(xExecute:= FALSE);
		close_file(xexecute:=FALSE);
 END_CASE
END_IF

IF xError THEN
	CASE FileError OF
		0: StrError:='';
		5100: StrError:=concat(INT_TO_STRING(FileError), ' First Error');
		5101: StrError:=concat(INT_TO_STRING(FileError), ' TIME_OUT'); 
		5102: StrError:=concat(INT_TO_STRING(FileError), ' ABORT');  
		5103: StrError:=concat(INT_TO_STRING(FileError), ' HANDLE_INVALID'); 
		5104: StrError:=concat(INT_TO_STRING(FileError), ' FILE NOT EXIST'); 
		5105: StrError:=concat(INT_TO_STRING(FileError), ' EXIST'); 
		5106: StrError:=concat(INT_TO_STRING(FileError), ' NO_MORE_ENTRIES'); 
		5107: StrError:=concat(INT_TO_STRING(FileError), ' NOT_EMPTY'); 
		5108: StrError:=concat(INT_TO_STRING(FileError), ' READ_ONLY_CAA');
		5109: StrError:=concat(INT_TO_STRING(FileError), ' WRONG_PARAMETR'); 
		5110: StrError:=concat(INT_TO_STRING(FileError), ' ERROR_UNKNOWN'); 
		5111: StrError:=concat(INT_TO_STRING(FileError), ' WRITE_INCOMPLETE'); 
		5112: StrError:=concat(INT_TO_STRING(FileError), ' FILE_NOT_IMPLEMENTED');
		5150: StrError:=concat(INT_TO_STRING(FileError), ' FIRST_MF');
		5199: StrError:=concat(INT_TO_STRING(FileError), ' LAST_ERROR');
		ELSE StrError:=concat(INT_TO_STRING(FileError), 'Unknow Error. Recomend reboot the system');
	END_CASE
ELSE
	StrError:='';
END_IF

END_PROGRAM

// Device/Application/READ_FILE_ON_SD
PROGRAM READ_FILE_ON_SD
VAR
	open_file			: FILE.Open;
	read_file			: FILE.Read;
	close_file			: FILE.Close;
	set_pos				: FILE.SetPos;
	get_size			: FILE.GetSize;
	get_attribute		: FILE.GetAttribute;
	
	RESET_FUNC			: WORD;
	RESET_SUC			: BOOL;
	FULL_NAME_OF_FILE   : STRING(255):='1';//Example /mnt/ufs/media/mmcblk0p1/Archive/AlaxAkbar.txt
	NAME_DIR			: STRING(255);
	size_name		    : WORD;
	ptr_name			: POINTER TO BYTE;
	START_STOP_READ		: WORD;
	cnt_cycle			: WORD;	
	i					: WORD;
	state_read			: BYTE;
	end_line_point		: UDINT;
	left_bytes			: UDINT;
	size_file			: UDINT;
	SIZE_HR				: WORD;
	SIZE_LR				: WORD;
	ptr_word			: POINTER TO WORD;
	read_sz				: UDINT;
	
END_VAR

IF RESET_FUNC=1 THEN
	state_read:=0;
	cnt_cycle:=1;
	open_file(xexecute:=FALSE);
	get_size(xexecute:=FALSE);
	read_file(xexecute:=FALSE);		
	close_file(xexecute:=FALSE);
	set_pos(xexecute:=FALSE);
	FOR i:=0 TO 124 DO
		buffer_wr[i]:=0;
	END_FOR
	RESET_SUC:=TRUE;
ELSE
	RESET_SUC:=FALSE;	
END_IF

IF START_STOP_READ=1 THEN
	READING:=TRUE;
END_IF

IF START_STOP_READ=0 THEN
	cnt_cycle:=0;
	READING:=FALSE;
	FOR i:=0 TO 124 DO
		buffer[i]:=0;
	END_FOR
END_IF

IF READING AND cnt_cycle=0 THEN

CASE state_read OF
		0:
		size_name:=%IW146;
		ptr_name:=ADR(FULL_NAME_OF_FILE);
		FOR i:=1 TO size_name DO
			ptr_name[i-1]:=WORD_TO_BYTE(buffer_name_file[i]);
		END_FOR		
		NAME_DIR:=SEL(%IW0=1,ProgramFiles,ArchiveFiles);//FALSE - ProgramFiles, TRUE - ArchiveFiles
		FULL_NAME_OF_FILE:=concat(NAME_DIR,FULL_NAME_OF_FILE);
		state_read:=1;
		
		1:
		open_file(
		xExecute:=TRUE , 
		xDone=> , 
		xBusy=> , 
		xError=> ExError, 
		sFileName:=FULL_NAME_OF_FILE, 
		eFileMode:=file.MODE.MREAD, 
		xExclusive:=, 
		eError=> FileError, 
		hFile=> );
		
		IF open_file.xDone THEN
			state_read:=2;
			end_line_point:=0;
		END_IF
		
		IF open_file.xError THEN
			IF FileError = 5104 THEN(*File not exist*)
				cnt_cycle:=1;
				open_file(xExecute:=FALSE);
			ELSE
				state_read:=5;	
			END_IF
			size_file:=0;
		END_IF
		
		2:
		get_size(
			xExecute:= TRUE, 
			xDone=> , 
			xBusy=> , 
			xError=> ExError, 
			sFileName:=FULL_NAME_OF_FILE , 
			eError=> FileError, 
			szSize=>left_bytes);
			
		IF get_size.xDone THEN
			state_read:=3;
			get_size(xExecute:= FALSE);
			size_file:=left_bytes;
			ptr_word:=ADR(size_file);
			SIZE_LR:=ptr_word[0];
			SIZE_HR:=ptr_word[1];
			IF left_bytes>250 THEN
				read_sz:=250;
			ELSE
				read_sz:=size_file;
			END_IF
			
		END_IF
		
		IF get_size.xError THEN
			state_read:=5;
		END_IF
			
		3:
		read_file(
			xExecute:=TRUE , 
			xAbort:= , 
			udiTimeOut:= , 
			xDone=> , 
			xBusy=> , 
			xError=> ExError, 
			xAborted=> , 
			hFile:=open_file.hFile , 
			pBuffer:=ADR(buffer), 
			szBuffer:=read_sz,
			szSize=>, 
			eError=> FileError);
			
		IF read_file.xDone  THEN
			state_read:=4;
			read_file(xExecute:= FALSE);
			end_line_point:=end_line_point+read_sz;
			IF left_bytes>250 THEN
				left_bytes:=left_bytes-250;
			END_IF
				
		END_IF
		
		IF read_file.xError THEN
			state_read:=5;
		END_IF
		
		4:
		set_pos(
			xExecute:= TRUE, 
			xDone=> , 
			xBusy=> , 
			xError=> ExError, 
			hFile:=open_file.hFile , 
			udiPos:=end_line_point , 	
			eError=>FileError);
		IF set_pos.xDone THEN
			set_pos(xExecute:= FALSE);
			IF left_bytes>0 THEN
				state_read:=3;
				cnt_cycle:=cnt_cycle+1;
			ELSE
				state_read:=5;
				cnt_cycle:=0;
			END_IF
			
			IF left_bytes<=250 THEN
				read_sz:=left_bytes;
				left_bytes:=0;
			END_IF
		END_IF
		
		IF set_pos.xError THEN
			state_read:=5;
		END_IF	
		
		5:
		close_file(
			xExecute:=TRUE , 
			xDone=> , 
			xBusy=> , 
			xError=> ExError, 
			hFile:=open_file.hFile , 
			eError=> FileError);
		
		IF close_file.xDone THEN
			state_read:=0;
			cnt_cycle:=cnt_cycle+1;
			open_file(xexecute:=FALSE);
			close_file(xexecute:=FALSE);
			FOR i:=0 TO 124 DO
				buffer_wr[i]:=0;
			END_FOR	
		END_IF
		
		IF close_file.xError THEN
			state_read:=5;
		END_IF	
			
 END_CASE
	
END_IF

IF ExError THEN
	CASE FileError OF
		0: StrError:='';
		5100: StrError:=concat(INT_TO_STRING(FileError), ' First Error');
		5101: StrError:=concat(INT_TO_STRING(FileError), ' TIME_OUT'); 
		5102: StrError:=concat(INT_TO_STRING(FileError), ' ABORT');  
		5103: StrError:=concat(INT_TO_STRING(FileError), ' HANDLE_INVALID'); 
		5104: StrError:=concat(INT_TO_STRING(FileError), ' FILE NOT EXIST'); 
		5105: StrError:=concat(INT_TO_STRING(FileError), ' EXIST'); 
		5106: StrError:=concat(INT_TO_STRING(FileError), ' NO_MORE_ENTRIES'); 
		5107: StrError:=concat(INT_TO_STRING(FileError), ' NOT_EMPTY'); 
		5108: StrError:=concat(INT_TO_STRING(FileError), ' READ_ONLY_CAA');
		5109: StrError:=concat(INT_TO_STRING(FileError), ' WRONG_PARAMETR'); 
		5110: StrError:=concat(INT_TO_STRING(FileError), ' ERROR_UNKNOWN'); 
		5111: StrError:=concat(INT_TO_STRING(FileError), ' WRITE_INCOMPLETE'); 
		5112: StrError:=concat(INT_TO_STRING(FileError), ' FILE_NOT_IMPLEMENTED');
		5150: StrError:=concat(INT_TO_STRING(FileError), ' FIRST_MF');
		5199: StrError:=concat(INT_TO_STRING(FileError), ' LAST_ERROR');
	END_CASE
ELSE
	StrError:='';
END_IF

END_PROGRAM

// Device/Application/WRITE_FILE_ON_SD
PROGRAM WRITE_FILE_ON_SD
VAR
	
	open_file			: FILE.Open;
	write_to_file		: FILE.Write;
	close_file			: FILE.Close;
	set_pos				: FILE.SetPos;
	get_size			: FILE.GetSize;
	
	FULL_NAME_OF_FILE	: STRING;
	size_name			: WORD;
	START_STOP_WRITE    : WORD;
	cnt_cycle			: BYTE;
	i 					: WORD;
	ptr_name			: POINTER TO BYTE;
	state_write			: BYTE;
	size_file			: UDINT;
	size_block			: WORD;
	iterator			: UDINT;
	CycleWriteDone		: WORD;	
END_VAR

IF START_STOP_WRITE=1 THEN
	WRITING:=TRUE;
END_IF

IF START_STOP_WRITE=0 THEN
	cnt_cycle:=0;
	WRITING:=FALSE;
	CycleWriteDone:=0;
END_IF

IF WRITING AND cnt_cycle=0 THEN
	CASE state_write OF
		0:
		size_name:=%IW146;
		ptr_name:=ADR(FULL_NAME_OF_FILE);
		FOR i:=0 TO size_name DO
			ptr_name[i]:=WORD_TO_BYTE(buffer_name_file[i]);
		END_FOR
		state_write:=1;
		cnt_cycle:=1;		
		
		1:
		open_file(
		xExecute:=TRUE , 
		xDone=> , 
		xBusy=> , 
		xError=> ExError, 
		sFileName:=concat('/mnt/ufs/media/mmcblk0p1/',FULL_NAME_OF_FILE), 
		eFileMode:=file.MODE.MWRITE, 
		xExclusive:=, 
		eError=> FileError, 
		hFile=> );
		
		IF open_file.xDone THEN
			state_write:=2;
		END_IF
			
		2:
		write_to_file(
			xExecute:=TRUE , 
			xAbort:= , 
			udiTimeOut:= , 
			xDone=> , 
			xBusy=> , 
			xError=> ExError, 
			xAborted=> , 
			hFile:=open_file.hFile , 
			pBuffer:= ADR(buffer_wr), 
			szSize:= size_block, 
			eError=> FileError);
 	
		IF write_to_file.xDone  THEN
			state_write:=3;
			write_to_file(xExecute:= FALSE);
			iterator:=iterator+size_block;	
		END_IF
		
		3:
		set_pos(
			xExecute:= TRUE, 
			xDone=> , 
			xBusy=> , 
			xError=> ExError, 
			hFile:=open_file.hFile , 
			udiPos:=iterator , 	
			eError=>FileError);
		IF set_pos.xDone THEN
			IF size_block<>242 THEN
				state_write:=4;
				cnt_cycle:=0;
			ELSE
				state_write:=2;
				cnt_cycle:=cnt_cycle+1;
			END_IF			
			set_pos(xExecute:= FALSE);
			CycleWriteDone:=1;
		END_IF
		
		4:
		close_file(
			xExecute:=TRUE , 
			xDone=> , 
			xBusy=> , 
			xError=> ExError, 
			hFile:=open_file.hFile , 
			eError=> FileError);
		
		IF close_file.xDone THEN
			state_write:=0;
			cnt_cycle:=cnt_cycle+1;
			open_file(xexecute:=FALSE);
			close_file(xexecute:=FALSE);	
		END_IF
			
 END_CASE
END_IF

IF ExError THEN
	CASE FileError OF
		0: StrError:='';
		5100: StrError:=concat(INT_TO_STRING(FileError), ' First Error');
		5101: StrError:=concat(INT_TO_STRING(FileError), ' TIME_OUT'); 
		5102: StrError:=concat(INT_TO_STRING(FileError), ' ABORT');  
		5103: StrError:=concat(INT_TO_STRING(FileError), ' HANDLE_INVALID'); 
		5104: StrError:=concat(INT_TO_STRING(FileError), ' FILE NOT EXIST'); 
		5105: StrError:=concat(INT_TO_STRING(FileError), ' EXIST'); 
		5106: StrError:=concat(INT_TO_STRING(FileError), ' NO_MORE_ENTRIES'); 
		5107: StrError:=concat(INT_TO_STRING(FileError), ' NOT_EMPTY'); 
		5108: StrError:=concat(INT_TO_STRING(FileError), ' READ_ONLY_CAA');
		5109: StrError:=concat(INT_TO_STRING(FileError), ' WRONG_PARAMETR'); 
		5110: StrError:=concat(INT_TO_STRING(FileError), ' ERROR_UNKNOWN'); 
		5111: StrError:=concat(INT_TO_STRING(FileError), ' WRITE_INCOMPLETE'); 
		5112: StrError:=concat(INT_TO_STRING(FileError), ' FILE_NOT_IMPLEMENTED');
		5150: StrError:=concat(INT_TO_STRING(FileError), ' FIRST_MF');
		5199: StrError:=concat(INT_TO_STRING(FileError), ' LAST_ERROR');
	END_CASE
ELSE
	StrError:='';
END_IF

END_PROGRAM

// Device/Application/Archive_manager
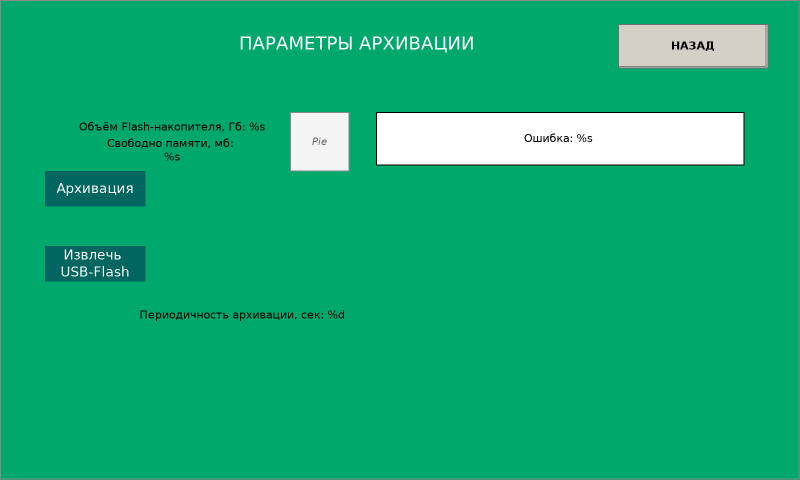
VISUALIZATION Archive_manager  // 800x480
    Textfield (227,26 260x35), "ПАРАМЕТРЫ АРХИВАЦИИ"
    Button (618,24 150x44), "НАЗАД"
        OnMouseClick:  Assign=Regim_choice, Type=Assignment
    Ellipse (290,112 59x59)
    Pie (290,112 59x59)
        p2124672552: Archive.memory_free_rotate
    Rectangle (35,117 274x20), "Объём Flash-накопителя, Гб: %s", text variable: Archive.memory_all
    Rectangle (35,137 274x26), "Свободно памяти, мб: %s", text variable: Archive.memory_used
    Rectangle (44,305 304x20), "Периодичность архивации, сек: %d", text variable: Archive.Arch_timout
        OnMouseClick: write the text variable via VisuDialogs.Numpad
    Rectangle (45,171 100x35), "Архивация", colour toggle: Archive.arch_en
        toggle Archive.arch_en
    Rectangle (45,246 100x35), "Извлечь USB-Flash", invisible if: Archive.memory_all_word=0
        OnMouseClick: execute { Archive.unmount:=true; }
    Rectangle (376,112 368x53), "Ошибка: %s", text variable: GVL.StrError
END_VISUALIZATION

// Device/Application/Center_indukt
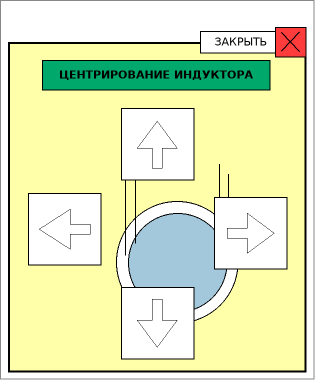
VISUALIZATION Center_indukt  // 315x380
    RoundedRectangle (8,42 298x330)
    Group (116,164 81x110)
        Ellipse (0,37 122x122)
        Ellipse (12,49 99x99)
        Group (9,0 104x66)
            Line (94,0) (94,79)
            Line (10,0) (10,79)
            Line (103,10) (103,90)
            Line (0,10) (0,91)
    Line (297,277)
    RoundedRectangle (121,287 73x72), colour toggle: PLC_PRG.CENTER_DOWN
        OnMouseUp: execute {  }
        OnMouseDown: execute {  }
    Polygon (137,320) (157,347) (177,320) (162,320) (162,299) (152,299) (152,320), colour toggle: PLC_PRG.CENTER_DOWN
        OnMouseDown: execute {  }
    InvisibleInput (109,278 95x90)
        OnMouseDown: execute { PLC_PRG.CENTER_DOWN := 1; }
        OnMouseUp: execute { PLC_PRG.CENTER_DOWN := 0; }
    RoundedRectangle (214,197 73x72), colour toggle: PLC_PRG.CENTER_RIGHT
        OnMouseUp: execute {  }
        OnMouseDown: execute {  }
    RoundedRectangle (121,108 73x72), colour toggle: PLC_PRG.CENTER_UP
        OnMouseUp: execute {  }
    Polygon (137,148) (157,121) (177,148) (162,148) (162,168) (152,168) (152,148), colour toggle: PLC_PRG.CENTER_UP
        OnMouseDown: execute {  }
    InvisibleInput (109,99 95x90)
        OnMouseDown: execute { PLC_PRG.CENTER_UP:=TRUE; }
        OnMouseUp: execute { PLC_PRG.CENTER_UP := FALSE; }
    Polygon (247,253) (274,233) (247,213) (247,228) (227,228) (227,238) (247,238), colour toggle: PLC_PRG.CENTER_RIGHT
        OnMouseDown: execute {  }
    InvisibleInput (202,188 95x90)
        OnMouseDown: execute { PLC_PRG.CENTER_RIGHT := 1; }
        OnMouseUp: execute { PLC_PRG.CENTER_RIGHT := 0; }
    RoundedRectangle (28,193 73x72), colour toggle: PLC_PRG.CENTER_LEFT
        OnMouseUp: execute {  }
        OnMouseDown: execute {  }
    Polygon (70,249) (39,229) (70,209) (70,224) (90,224) (90,234) (70,234), colour toggle: PLC_PRG.CENTER_LEFT
        OnMouseDown: execute {  }
    InvisibleInput (18,188 95x90)
        OnMouseDown: execute { PLC_PRG.CENTER_LEFT := 1; }
        OnMouseUp: execute { PLC_PRG.CENTER_LEFT := 0; }
    Textfield (42,60 228x30), "ЦЕНТРИРОВАНИЕ ИНДУКТОРА"
    Line (289,21)
    Group (200,27 106x30)
        OnMouseClick:  Dialog=Center_indukt, Result=OK, NumpadKeypadSet=True
        Rectangle (0,4 82x22), "ЗАКРЫТЬ"
        RoundedRectangle (75,0 31x30)
        Line (99,5) (81,24)
        Line (81,5) (99,24)
    InvisibleInput (178,9 157x66)
        OnMouseClick:  Dialog=Center_indukt, Result=OK, NumpadKeypadSet=True
END_VISUALIZATION

